// ---- 20_Product/10_BCF/11_Conv/15_Subsystem/10_Helper/F_GetSubSystemExternErrorData.TcPOU
FUNCTION F_GetSubSystemExternErrorData : ST_ErrorDataSet
(**************************************************************************************
 * 	Application		:	BoxControl Framework
 *	Revision		:	$Revision: 404529 $
 *	Revision date	:	$Date: 2018-04-23 08:21:38 +0200 (Mo., 23 Apr 2018) $
 *	Last changed by	:	$Author: b7bolm $
 *	URL				:	$URL: http://almscdc.swisslog.com/repo/SWPD/Development/BoxControlFramework/20_Release/trunk/01_Software/BCF/BCF/JumpStart/20_Product/10_App/15_Subsystem/10_Lib/10_Conv/10_Functions/F_GetSubSystemExternErrorData.TcPOU $
 *
 *	Purpose			:	Return subsystem error data
 *
 * ------------------------------------------------------------------------------------
 *	Copyright Swisslog [IP AG], Switzerland. All rights reserved.
 * 
 * ------------------------------------------------------------------------------------
 *	
 * 	Revision History: 
 *
 * 	VERSION			DATE			INITIALS			DESCRIPTION
 *	0.1				01.01.2001		swl					Example
 *
 **************************************************************************************)


// Check reference is valid
IF __ISVALIDREF(Subsystemregistry.rSubsystemData) THEN
	// Return error data
	F_GetSubSystemExternErrorData :=Subsystemregistry.rSubsystemData.ErrorData.ExternalError;
END_IF

END_FUNCTION

// ---- 20_Product/10_BCF/11_Conv/15_Subsystem/10_Helper/F_GetSubSystemInterface.TcPOU
FUNCTION F_GetSubsystemInterface : ST_SubsystemInterface
(**************************************************************************************
 * 	Application		:	BoxControl Framework
 *	Revision		:	$Revision: 404529 $
 *	Revision date	:	$Date: 2018-04-23 08:21:38 +0200 (Mo., 23 Apr 2018) $
 *	Last changed by	:	$Author: b7bolm $
 *	URL				:	$URL: http://almscdc.swisslog.com/repo/SWPD/Development/BoxControlFramework/20_Release/trunk/01_Software/BCF/BCF/JumpStart/20_Product/10_App/15_Subsystem/10_Lib/10_Conv/10_Functions/F_GetSubSystemInterface.TcPOU $
 *
 *	Purpose			:	Returns group interface
 *
 * ------------------------------------------------------------------------------------
 *	Copyright Swisslog [IP AG], Switzerland. All rights reserved.
 * 
 * ------------------------------------------------------------------------------------
 *	
 * 	Revision History: 
 *
 * 	VERSION			DATE			INITIALS			DESCRIPTION
 *	0.1				01.01.2001		swl					Example
 *
 **************************************************************************************)

// Get Master speed from subsystem
IF __ISVALIDREF(SubsystemRegistry.rSubsystem) THEN
	// Return Subsystem interface
	F_GetSubsystemInterface := SubsystemRegistry.rSubsystem.SubsystemInterface;
END_IF

END_FUNCTION

// ---- 20_Product/10_BCF/11_Conv/15_Subsystem/10_Helper/F_GetSubSystemSettings.TcPOU
FUNCTION F_GetSubsystemSettings : ST_CFG_Subsystem
(**************************************************************************************
 * 	Application		:	BoxControl Framework
 *	Revision		:	$Revision: 404529 $
 *	Revision date	:	$Date: 2018-04-23 08:21:38 +0200 (Mo., 23 Apr 2018) $
 *	Last changed by	:	$Author: b7bolm $
 *	URL				:	$URL: http://almscdc.swisslog.com/repo/SWPD/Development/BoxControlFramework/20_Release/trunk/01_Software/BCF/BCF/JumpStart/20_Product/10_App/15_Subsystem/10_Lib/10_Conv/10_Functions/F_GetSubSystemSettings.TcPOU $
 *
 *	Purpose			:	Returns group settings
 *
 * ------------------------------------------------------------------------------------
 *	Copyright Swisslog [IP AG], Switzerland. All rights reserved.
 * 
 * ------------------------------------------------------------------------------------
 *	
 * 	Revision History: 
 *
 * 	VERSION			DATE			INITIALS			DESCRIPTION
 *	0.1				01.01.2001		swl					Example
 *
 **************************************************************************************)
VAR
	SubsystemReg	: ST_SubsystemRegistryConv;
END_VAR


// Get Master speed from subsystem
IF __ISVALIDREF(SubsystemRegistry.rSettingsSubsystem) THEN
	// Return Subsystem settings
	F_GetSubsystemSettings := SubsystemRegistry.rSettingsSubsystem;
END_IF

END_FUNCTION

// ---- 20_Product/10_BCF/11_Conv/15_Subsystem/10_Helper/F_ResetExternalSubsystemError.TcPOU
FUNCTION F_ResetExternalSubsystemError : BOOL
(**************************************************************************************
 * 	Application		:	BoxControl Framework
 *	Revision		:	$Revision: 404529 $
 *	Revision date	:	$Date: 2018-04-23 08:21:38 +0200 (Mo., 23 Apr 2018) $
 *	Last changed by	:	$Author: b7bolm $
 *	URL				:	$URL: http://almscdc.swisslog.com/repo/SWPD/Development/BoxControlFramework/20_Release/trunk/01_Software/BCF/BCF/JumpStart/20_Product/10_App/15_Subsystem/10_Lib/10_Conv/10_Functions/F_ResetExternalSubsystemError.TcPOU $
 *
 *	Purpose			:	Reset external error
 *						Add an External error, which will be reported over the configured
 *						position.
 *						
 *
 * ------------------------------------------------------------------------------------
 *	Copyright Swisslog [IP AG], Switzerland. All rights reserved.
 * 
 * ------------------------------------------------------------------------------------
 *	
 * 	Revision History: 
 *
 * 	VERSION			DATE			INITIALS			DESCRIPTION
 *	0.1				01.01.2001		swl					Example
 *
 **************************************************************************************)
VAR_INPUT
	Reset			: BOOL;
END_VAR


IF __ISVALIDREF(SubsystemRegistry.rSubsystem) THEN
	// Reset external error on instance
	SubsystemRegistry.rSubsystem.M_ResetExternalError(
		mReset := Reset);
END_IF

END_FUNCTION

// ---- 20_Product/10_BCF/11_Conv/15_Subsystem/10_Helper/F_ResetSubsystemError.TcPOU
FUNCTION F_ResetSubsystemError : BOOL
(**************************************************************************************
 * 	Application		:	BoxControl Framework
 *	Revision		:	$Revision: 404529 $
 *	Revision date	:	$Date: 2018-04-23 08:21:38 +0200 (Mo., 23 Apr 2018) $
 *	Last changed by	:	$Author: b7bolm $
 *	URL				:	$URL: http://almscdc.swisslog.com/repo/SWPD/Development/BoxControlFramework/20_Release/trunk/01_Software/BCF/BCF/JumpStart/20_Product/10_App/15_Subsystem/10_Lib/10_Conv/10_Functions/F_ResetSubsystemError.TcPOU $
 *
 *	Purpose			:	Reset Subsystem error
 *
 * ------------------------------------------------------------------------------------
 *	Copyright Swisslog [IP AG], Switzerland. All rights reserved.
 * 
 * ------------------------------------------------------------------------------------
 *	
 * 	Revision History: 
 *
 * 	VERSION			DATE			INITIALS			DESCRIPTION
 *	0.1				01.01.2001		swl					Example
 *
 **************************************************************************************)

// Reset subsystem error
IF __ISVALIDREF(SubsystemRegistry.rSubsystem) THEN
	// Reset error on Subsystem
	SubsystemRegistry.rSubsystem.M_ResetError();
END_IF

END_FUNCTION

// ---- 20_Product/10_BCF/11_Conv/15_Subsystem/10_Helper/F_SetExternalSubsystemError.TcPOU
FUNCTION F_SetExternalSubsystemError : BOOL
(**************************************************************************************
 * 	Application		:	BoxControl Framework
 *	Revision		:	$Revision: 404529 $
 *	Revision date	:	$Date: 2018-04-23 08:21:38 +0200 (Mo., 23 Apr 2018) $
 *	Last changed by	:	$Author: b7bolm $
 *	URL				:	$URL: http://almscdc.swisslog.com/repo/SWPD/Development/BoxControlFramework/20_Release/trunk/01_Software/BCF/BCF/JumpStart/20_Product/10_App/15_Subsystem/10_Lib/10_Conv/10_Functions/F_SetExternalSubsystemError.TcPOU $
 *
 *	Purpose			:	Set external error
 *						Add an External error, which will be reported over the configured
 *						position.
 *						
 *
 * ------------------------------------------------------------------------------------
 *	Copyright Swisslog [IP AG], Switzerland. All rights reserved.
 * 
 * ------------------------------------------------------------------------------------
 *	
 * 	Revision History: 
 *
 * 	VERSION			DATE			INITIALS			DESCRIPTION
 *	0.1				01.01.2001		swl					Example
 *
 **************************************************************************************)
VAR_INPUT
	ErrorType		: E_ErrorType; // Error message type
	ErrorParam		: STRING(System.ERROR_PARAM_STRINGLENGTH); // Error parameter
	ErrorMsg		: INT; // Error message as String (Will be mapped to error code)
END_VAR


IF __ISVALIDREF(SubsystemRegistry.rSubsystem) THEN
	// Set external error on instance
	SubsystemRegistry.rSubsystem.M_SetExternalError(
		mErrorType 	:= ErrorType,
		mErrorParam := ErrorParam,
		mErrorCode 	:= ErrorMsg);
END_IF

END_FUNCTION

// ---- 20_Product/20_ProBox/10_Base/09_Overrides/FB_PB_FunctionConv.TcPOU
FUNCTION_BLOCK INTERNAL FB_PB_FunctionConv EXTENDS FB_FunctionConv
VAR_INPUT
END_VAR
VAR_OUTPUT
END_VAR

METHOD PROTECTED M_GetNextTransportData : REFERENCE TO ST_TransportData

VAR_INPUT
	mZoneNumber 	: INT; // Number of the zone
END_VAR

VAR
	NextFunction	: E_FunctionNumber;
	TempCopy		: E_FunctionNumber;
END_VAR

//Solves BCFD-11487 M_GetTransportData returns TransportData for wrong zone (in some situations)
//Solves BCFD-11583 HandoverState enters Active when next is Taking over from another function

//when Next function transport data is expected, we need to make sure that M_GetNextTransportData return correct data (Next -> Previus)
NextFunction := FunctionInterface.In.eNextFunctionNumber;
IF(__ISVALIDREF(FunctionRegistry[NextFunction].rFunctionInterface)) THEN
	TempCopy := FunctionRegistry[NextFunction].rFunctionInterface.In.eNextFunctionNumber;
	FunctionRegistry[NextFunction].rFunctionInterface.In.eNextFunctionNumber := E_FunctionNumber.F_BEGIN_FUNCTION;
	M_GetNextTransportData REF= SUPER^.M_GetNextTransportData(mZoneNumber);
	FunctionRegistry[NextFunction].rFunctionInterface.In.eNextFunctionNumber := TempCopy;
ELSE
	M_GetNextTransportData REF= SUPER^.M_GetNextTransportData(mZoneNumber);
END_IF
END_METHOD

METHOD PROTECTED M_GetPreviousTransportData: REFERENCE TO ST_TransportData

VAR_INPUT
	mZoneNumber 	: INT; // Number of the zone
END_VAR

VAR
	PrevFunction	: E_FunctionNumber;
	TempCopy		: E_FunctionNumber;
END_VAR

//Solves BCFD-11487 M_GetTransportData returns TransportData for wrong zone (in some situations)
//Solves BCFD-11583 HandoverState enters Active when next is Taking over from another function

//when previous function transport data is expected, we need to make sure that M_GetNextTransportData return correct data (prevous ->Next)
PrevFunction := FunctionInterface.In.ePrevFunctionNumber;
IF(__ISVALIDREF(FunctionRegistry[PrevFunction].rFunctionInterface)) THEN
	TempCopy := FunctionRegistry[PrevFunction].rFunctionInterface.In.ePrevFunctionNumber;
	FunctionRegistry[PrevFunction].rFunctionInterface.In.ePrevFunctionNumber := E_FunctionNumber.F_BEGIN_FUNCTION;
	M_GetPreviousTransportData REF= SUPER^.M_GetPreviousTransportData(mZoneNumber);
	FunctionRegistry[PrevFunction].rFunctionInterface.In.ePrevFunctionNumber := TempCopy;
ELSE
	M_GetPreviousTransportData REF= SUPER^.M_GetPreviousTransportData(mZoneNumber);
END_IF
END_METHOD

END_FUNCTION_BLOCK

// ---- 20_Product/20_ProBox/22_ProMove/03_Controls/02_TransportControl/FB_PB_TransportControlEmulation.TcPOU
FUNCTION_BLOCK FB_PB_TransportControlEmulation EXTENDS FB_TransportControlEmulation
(**************************************************************************************
 * 	Application		:	Pro Box
 *	Revision		:	$Revision:  $
 *	Revision date	:	$Date: $
 *	Last changed by	:	$Author: q8hedls $
 *	URL				:	$$
 *
 *	Purpose			:	Override BCF Transport control emulation
 *
 * ------------------------------------------------------------------------------------
 *	Copyright Swisslog [IP AG], Switzerland. All rights reserved.
 * 
 * ------------------------------------------------------------------------------------
 *	
 **************************************************************************************)
VAR_INPUT
	
END_VAR

VAR_IN_OUT
	//ZoneData				: ST_ZoneDataEmulation; // Zone data
END_VAR


SUPER^(ZoneData :=ZoneData);

END_FUNCTION_BLOCK

// ---- 20_Product/20_ProBox/22_ProMove/03_Controls/02_TransportControl/FB_ProBoxTransportControl.TcPOU
//ProBox transportcontroller
FUNCTION_BLOCK FB_ProBoxTransportControl EXTENDS FB_TransportControl
(**************************************************************************************
 * 	Application		:	ProBox
 *	Revision		:	$Revision:  $
 *	Revision date	:	$Date: $
 *	Last changed by	:	$Author: $
 *	URL				:	$URL: $
 *
 *	Purpose			:	The transport control is responsible for the coordinated
 *                      physical TU and logical data movement and ensures the relation
 *                      to the position for the ProMove Pallet system.
 *
 **************************************************************************************)
VAR_INPUT
	CtrlInPbTc				: ST_CtrlInPbTc;// Control input for Pro box Transport control
END_VAR
VAR	
	_PB_TransportCtrlData	: ST_PB_TransportCtrl;
	_ValidPrevFunction		: E_FunctionNumber;
	_ValidPrevZone			: INT;	
	_PbTcDebugLogLevel		: INT:=0; 		//ProBox Transport Control Debug level. 0 = Off, 1=States, 2 Verbose
END_VAR

VAR_TEMP
		
	PB_SimultaniousDisableTakeover		 :BOOL;	//TRUE = Release TU's
	PB_PreventTakeover					: BOOL; //For Multi Zone Functions
	PB_PreventHandover					: BOOL; //workaround for BCF transportcontroller not capable of handling a occupied after transition error
	PB_InhibitHandoverRun				: BOOL;	//Force stopping of drive
	PB_ForceTakeoverRun					: BOOL; //Force motor run of drive
	
	// internal variables only for debuging purposes
	PrevTrspState						: E_TransportState;
	PrevHandOvrState					: E_HandOverState;
	PrevTakeOvrState					: E_TakeOverState;		
END_VAR

IF(_PbTcDebugLogLevel>0) THEN
	// internal variables onlyfor debuging purposes
	PrevTrspState := ZoneData.TransportControlData.eTransportState;
	PrevHandOvrState := ZoneData.TransportControlData.eHandOverState;
	PrevTakeOvrState := ZoneData.TransportControlData.eTakeOverState;
END_IF

//---------------------------------------------------------------------------------------------------
// Init and checks for ProBox
//---------------------------------------------------------------------------------------------------
_M_PB_Init(ZoneData);
_M_InputMapping();


//---------------------------------------------------------------------------------------------------
// Pre-tasks that must be performed before runnign BCF transportcontrol
//---------------------------------------------------------------------------------------------------

_M_SyntheticSensor(ZoneData);
_M_GapCheck(ZoneData,ErrorData);
_M_PB_PreErrorCheck(ZoneData,ErrorData,PB_PreventTakeover,PB_PreventHandover);
_M_PB_PreTrspCtrl(ZoneData,ErrorData,PB_ForceTakeoverRun,PB_SimultaniousDisableTakeover,PB_PreventTakeover);

//---------------------------------------------------------------------------------------------------
// Call BCF TransportController
//---------------------------------------------------------------------------------------------------

TransportEnableTakeOver := TransportEnableTakeOver AND (NOT PB_SimultaniousDisableTakeover AND NOT PB_PreventTakeover);
TransportEnableHandOver := TransportEnableHandOver AND NOT PB_PreventHandover;
SUPER^(ZoneData:=ZoneData,ErrorData:=ErrorData);



//---------------------------------------------------------------------------------------------------
// Post-tasks that must be performed after BCF transportcontrol where executed
//---------------------------------------------------------------------------------------------------
_M_PB_PostTrspCtrl(ZoneData,PB_InhibitHandoverRun);
_M_PB_PostErrorCheck(ZoneData);
_M_PB_SpeedControl(ZoneData);

//PB transportcontrol controlling driving.
Outputs.DriveHandoverRun := (Outputs.DriveHandoverRun AND NOT PB_InhibitHandoverRun);
Outputs.DriveTakeoverRun := Outputs.DriveTakeoverRun OR PB_ForceTakeoverRun;

ZoneData.TransportControlData.Stopped := Param.rOperationState.eState = E_PositionState.STOPPED OR
									 	 Param.rOperationState.eState = E_PositionState.STOPPING AND NOT
									     DriveTakeoverRun AND NOT DriveHandoverRun;

//check RequestNext / DeleteNext and RequestPrev / DeletePrev
_M_ControlTransportRequests();



//---------------------------------------------------------------------------------------------------
// log transitions (To be deleted
//---------------------------------------------------------------------------------------------------
IF(_PbTcDebugLogLevel>0) THEN
	IF( PrevTrspState<>ZoneData.TransportControlData.eTransportState OR 
		PrevHandOvrState<>ZoneData.TransportControlData.eHandOverState OR
		PrevTakeOvrState<>ZoneData.TransportControlData.eTakeOverState) THEN
					DebugMsg := F_AddDividerToSisString(Param.rSettings.ZoneName);				
					DebugMsg := CONCAT(DebugMsg, '. Transport state: ');
					DebugMsg := CONCAT(DebugMsg, INT_TO_STRING(ZoneData.TransportControlData.eTransportState));
					DebugMsg := CONCAT(DebugMsg, '. Handover state: ');
					DebugMsg := CONCAT(DebugMsg, INT_TO_STRING(ZoneData.TransportControlData.eHandOverState));
					DebugMsg := CONCAT(DebugMsg, '. Takeover state: ');
					DebugMsg := CONCAT(DebugMsg, INT_TO_STRING(ZoneData.TransportControlData.eTakeOverState));
					DebugMsg := CONCAT(DebugMsg, '. HO Run: ');
					DebugMsg := CONCAT(DebugMsg, BOOL_TO_STRING(Outputs.DriveHandoverRun));
					DebugMsg := CONCAT(DebugMsg, '. TO Run: ');
					DebugMsg := CONCAT(DebugMsg, BOOL_TO_STRING(Outputs.DriveTakeoverRun));				
					fbDebugMsg.M_SendInfoMsg(DebugMsg);
	END_IF	
END_IF

//---------------------------------------------------------------------------------------------------
// Set error param with informative descriptions 
//---------------------------------------------------------------------------------------------------
//Only set the ErrorParam once, ie when the zone has no error. Also, do not override ErrorParam if there is text already set
IF(ZoneData.ErrorData.ErrorState <> E_ErrorState.ERROR AND ErrorData.ErrorParam[0]=0) THEN
	
	CASE ErrorData.ErrorCode.Conv OF 
		E_ErrorConv.TIMEOUT_TAKEOVER:
			ErrorData.ErrorParam	:= 'Takeover abnormal distance(TimeOut)';		
		E_ErrorConv.POSITION_OCCUPIED_BEFORE_TAKEOVER:
        	ErrorData.ErrorParam	:= 'Position occupied before takeover';
		E_ErrorConv.POSITION_OCCUPIED_AFTER_HANDOVER:
			ErrorData.ErrorParam	:= 'Position occupied after transmission';		
		E_ErrorConv.TU_DATA_SET_EMPTY_ZONE_OCCUPIED:
			ErrorData.ErrorParam	:= 'TU data set empty, position occupied'; 
  		E_ErrorConv.TU_DATA_SET_OCCUPIED_ZONE_FREE:
			ErrorData.ErrorParam	:= 'TU data set occupied, position free';	
		
	END_CASE
	
END_IF

METHOD PRIVATE _M_AllZonesOccupied : BOOL
VAR_INPUT
END_VAR

_M_AllZonesOccupied := _M_CountTus() = _PB_TransportCtrlData.NumberOfZones;
END_METHOD

METHOD PRIVATE _M_CheckZoneError : BOOL
VAR_INPUT
	eFunctionNumber		: E_FunctionNumber; // Function number
	ZoneNumber			: INT; // Zone number
END_VAR
// Check if function number and zone is valid
IF eFunctionNumber > E_FunctionNumber.F_BEGIN_FUNCTION AND
   eFunctionNumber < E_FunctionNumber.F_END_FUNCTION AND
   ZoneNumber > 0 AND ZoneNumber <= NUMBER_OF_ZONES_PER_FUNCTION THEN
  
   IF __ISVALIDREF(FunctionRegistry[eFunctionNumber].Zone[ZoneNumber].refZoneData) THEN
		// Zone errordata
		_M_CheckZoneError := FunctionRegistry[eFunctionNumber].Zone[ZoneNumber].refZoneData.ErrorData.Error.ErrorType = E_ErrorType.ERROR;
	END_IF
END_IF
END_METHOD

METHOD PRIVATE _M_ControlTransportRequests : BOOL
VAR_INPUT
END_VAR
//Disable fbRoutingServiceRetry waiting for RECALL_SERVICE_TIMEOUT ie 2S to request next function.
IF(SUPER^.Init AND  Param.rSettings.EnableRoutingUpdate AND _PB_TransportCtrlData.NumberOfZones>1 AND _PB_TransportCtrlData.IsFirstZone) THEN
	fbRoutingServiceRetry(IN := TRUE);
END_IF



//PB-6238 eNextFunctionNumber not set to F_BEGIN_FUNCTION after pallet removal
//request next function required when a zone is in state free.
IF(_PB_TransportCtrlData.NumberOfZones>1 AND _PB_TransportCtrlData.IsLastZone) THEN
	{warning disable C0371}
	IF( ZoneData.TransportControlData.eTransportState = E_TransportState.FREE) THEN		
		Outputs.DeleteNextTransportData:=TRUE;// request next
	END_IF
	{warning restore C0371}
END_IF


// control Delete next transportdata for multi zone functions. Don't delete next transport data unless finished handover
// fix for BCFD-11642 - TransportControl M_RequestPrev deletes previous on the same cycle as the transport starts
// -Also single zone functions needs to reset reqest signals
IF(Outputs.DeleteNextTransportData AND NOT Outputs.RequestNextTransportData) THEN
	//DeleteNextTransportData is requested	
	IF(_M_TransferBusy(Param.ZoneNumber,3)) THEN		
		Outputs.DeleteNextTransportData:=FALSE;	//Prevent delete next function			
	END_IF	
END_IF
IF(Outputs.DriveHandoverRun) THEN (*PB-5879 - TransportControl - TransportUnit transport error	AND BCFD-11642 - TransportControl M_RequestPrev deletes previous on the same cycle as the transport starts*)
	Outputs.DeleteNextTransportData:=FALSE;	//Prevent delete next function
	Outputs.RequestNextTransportData:=FALSE;//Prevent delete next function
END_IF

// control Delete prev transportdata for multi zone functions. Don't delete Prev transport data unless all zones finished takeover
// -Also single zone functions needs to reset reqest signals 
IF(Outputs.DeletePrevTransportData AND NOT Outputs.RequestPrevTransportData) THEN
	//DeletePrevTransportData is requested	
	IF(_M_TransferBusy(Param.ZoneNumber,1)) THEN
		Outputs.DeletePrevTransportData:=FALSE;	//Prevent delete previous function		
	END_IF			
END_IF
// fix for BCFD-11642 - TransportControl M_RequestPrev deletes previous on the same cycle as the transport starts
IF(Outputs.DriveTakeoverRun) THEN	
	Outputs.DeletePrevTransportData:=FALSE;	//Prevent delete previous function
	Outputs.RequestPrevTransportData:=FALSE;	//Prevent delete previous function
END_IF
END_METHOD

METHOD PRIVATE _M_CountTus : INT
VAR
	i,OccupiedCount:INT;
END_VAR
//Count TU's
FOR i:=1 TO _PB_TransportCtrlData.NumberOfZones DO
	IF(__ISVALIDREF(FunctionRegistry[Param.reFunctionNumber].Zone[i].refZoneData)) THEN
		IF(FunctionRegistry[Param.reFunctionNumber].Zone[i].refZoneData.TransportControlData.Occupied) THEN
			OccupiedCount := OccupiedCount + 1;
		END_IF
	END_IF
END_FOR
	
_M_CountTus:=OccupiedCount;
END_METHOD

METHOD PRIVATE _M_GapCheck : BOOL
VAR_IN_OUT
	ZoneData				: ST_ZoneData;
	ErrorData 				: ST_ErrorDataSet; // Error data 
END_VAR
VAR_INST		
	GapCheckState			: INT;			
	distanceMeter			: FB_DisplacementMeter();
	TestRunning	: BOOL;
END_VAR
VAR
	QuitTest				: BOOL;
END_VAR
IF(_PB_TransportCtrlData.NumberOfZones=1 OR NOT _PB_TransportCtrlData.IsLastZone) THEN
	RETURN;
END_IF


//Escape test
QuitTest := ZoneData.TransportControlData.eTransportState <> E_TransportState.SIMULTANEOUS AND
			ZoneData.TransportControlData.eTransportState <> E_TransportState.SIMULTANEOUS_STOP; 

CASE  GapCheckState OF
	0:		
		//Start test
		IF( ZoneData.TransportControlData.eTakeOverState = E_TakeOverState.ACTIVE AND
			ZoneData.TransportControlData.eTransportState = E_TransportState.SIMULTANEOUS) THEN			
			GapCheckState := GapCheckState+1;
			TestRunning:=FALSE;
		END_IF
	1:
		//check time when sensor detects gap of rear edge
		IF(NOT ZoneOccupied) THEN
			TestRunning:=TRUE;
			GapCheckState := GapCheckState+1;			
		ELSIF(QuitTest) THEN
			GapCheckState:=0;
		END_IF
		
	2: //Check when new pallet arrives
		IF(ZoneOccupied) THEN
			IF(distanceMeter.Q) THEN				 
				GapCheckState := GapCheckState+1; //Test successful				
			ELSE
				GapCheckState :=4; //error state				
			END_IF
		ELSIF(QuitTest) THEN
			GapCheckState := GapCheckState+1;
		END_IF 
	
	3:	
		//wait for Escape test to occure.
		IF(QuitTest) THEN			
			GapCheckState:=0;
		END_IF 
	4:
		//error
		F_SetError(	
					ErrorType	:= E_ErrorType.ERROR,
					ErrorParam	:= 'Gap not detected',
					ErrorMsg	:= E_ErrorConv.GAP_CHECK_ACTIVE,
					ErrorData	:= ErrorData);		
					
		//recover from error. sensor needs to be un-occupied. (or should it be enought with just a acknowledge of error?)
		IF(NOT ZoneOccupied) THEN
			GapCheckState:=0;
		END_IF
		
END_CASE


distanceMeter(
	Run:=TestRunning, 
	EncoderValueInc:=SUPER^.EncoderValue,
	MaxEncoderValueInc 	:= SUPER^.MaxEncoderValue, 
	RateIncPerMM:=1,
	SetPoint := 100 (*mm*));
END_METHOD

METHOD PRIVATE _M_InputMapping : BOOL
VAR_INPUT
END_VAR
VAR
	ElementNumber : E_ElementNumber;
END_VAR

//Prerequsities for ProBox transports
IF(Param.rSettings.EnableMFC) THEN
	//Following parameters must have defined state in order for ProBox to guarantee known functionality
	Param.rSettings.EnableFreeRun := FALSE;
	Param.rSettings.EnableMultizone := FALSE;
	Param.rSettings.EnableJamAutoReset := FALSE;
	Param.rSettings.ClearingDistance := 0;
	Param.rSettings.AddTU_Data := FALSE;
	Param.rSettings.DeleteTU_DataTakeOver := FALSE;
	Param.rSettings.DeleteTU_DataZoneFree := FALSE;
	Param.rSettings.EnablePrestart:=FALSE;				//important to set to false for transfer units
	Param.rSettings.EnableRoutingUpdate:=TRUE;			//Default ON
END_IF

//Transport control Inputs
EnableFastSpeed:=FALSE;			//Probox needs an alternative way of treating low speeds than BCF transport control. (this functionality is always enabled, but the EnableFastSpeed is set to false so that the BCF transport controller shall not run code unnecessary


IF(__ISVALIDREF(FunctionRegistry[Param.reFunctionNumber].rFunctionInterface)) THEN
	IF(NOT FunctionRegistry[Param.reFunctionNumber].rFunctionInterface.In.FunctionEnable) THEN
		TransportEnableHandOver := FALSE;
		IF(_M_CountTus()=0 AND _PB_TransportCtrlData.IsFirstZone) THEN 
			TransportEnableTakeOver:=FALSE; //Disable takeover if all zones are free
		END_IF 
		TransportEnableHandOver:=FALSE; //disable handover for all zones
	END_IF
END_IF


IF(__ISVALIDREF(FunctionRegistry[Param.reFunctionNumber].rSettingsFunction)) THEN
	ElementNumber := FunctionRegistry[Param.reFunctionNumber].rSettingsFunction.eElementLink;
	IF(__ISVALIDREF(ElementRegistry[ElementNumber].rElementInterface)) THEN
		IF(NOT ElementRegistry[ElementNumber].rElementInterface.In.ElementEnable) THEN			
			IF(_M_CountTus()=0 AND _PB_TransportCtrlData.IsFirstZone) THEN 
				TransportEnableTakeOver:=FALSE; //Disable takeover if all zones are free
			END_IF
			TransportEnableHandOver:=FALSE; //disable handover for all zones
		END_IF	
	END_IF
END_IF
END_METHOD

// Check if zone is deslugging 
METHOD PRIVATE _M_IsDeslugging : BOOL
VAR_INPUT
END_VAR
VAR
	NextNumberOfZones : INT;
	MeNumberOfZones : INT;
	OccupiedCount:INT;
	IsLastZone : BOOL;
END_VAR

//Last zone shall check if deslugging
IF(NOT _PB_TransportCtrlData.IsLastZone) THEN
	RETURN;
END_IF

// Check if function number is valid
IF NextTransportData.eFunctionNumber > E_FunctionNumber.F_BEGIN_FUNCTION AND
   NextTransportData.eFunctionNumber < E_FunctionNumber.F_END_FUNCTION THEN
  	
	IF __ISVALIDREF(FunctionRegistry[NextTransportData.eFunctionNumber].rSettingsFunction) THEN   		
   		NextNumberOfZones := FunctionRegistry[NextTransportData.eFunctionNumber].rSettingsFunction.NumberOfZones;
	ELSE
		RETURN;		 
	END_IF
	
			
	//Count TU's on own function
	OccupiedCount := _M_CountTus();
			
	// Deslugging whait with handover last TU until next function has filled upp all zones.  
	_M_IsDeslugging := NextNumberOfZones < _PB_TransportCtrlData.NumberOfZones AND (OccupiedCount + NextNumberOfZones <= _PB_TransportCtrlData.NumberOfZones); 
	
END_IF
END_METHOD

METHOD _M_PB_Init : BOOL
VAR_IN_OUT
	ZoneData					: ST_ZoneData;
END_VAR

IF( NOT ZoneData.Init) THEN
	_PB_TransportCtrlData.Init:=FALSE;		
END_IF

IF(NOT _PB_TransportCtrlData.Init) THEN
	IF __ISVALIDREF(FunctionRegistry[Param.reFunctionNumber].rSettingsFunction) THEN   		
   		_PB_TransportCtrlData.NumberOfZones := FunctionRegistry[Param.reFunctionNumber].rSettingsFunction.NumberOfZones;
		_PB_TransportCtrlData.Init := TRUE; 
	END_IF
	//Set to Default value.
	MaxEncoderValue	:= 16#FFFF;
	
ELSE
	//For each call check following.
	IF __ISVALIDREF(FunctionRegistry[Param.reFunctionNumber].rSettingsFunction) THEN

		_PB_TransportCtrlData.IsFirstZone := (Param.ZoneNumber = 1 AND  FunctionRegistry[Param.reFunctionNumber].rSettingsFunction.FlowDirectionREV = FALSE) OR
											 (Param.ZoneNumber = _PB_TransportCtrlData.NumberOfZones AND  FunctionRegistry[Param.reFunctionNumber].rSettingsFunction.FlowDirectionREV = TRUE);   		
   		
		_PB_TransportCtrlData.IsLastZone := (Param.ZoneNumber = 1 AND  FunctionRegistry[Param.reFunctionNumber].rSettingsFunction.FlowDirectionREV = TRUE) OR
											 (Param.ZoneNumber = _PB_TransportCtrlData.NumberOfZones AND  FunctionRegistry[Param.reFunctionNumber].rSettingsFunction.FlowDirectionREV = FALSE);
		
		_PB_TransportCtrlData.LastZoneIx := SEL(NOT FunctionRegistry[Param.reFunctionNumber].rSettingsFunction.FlowDirectionREV ,1,_PB_TransportCtrlData.NumberOfZones);
   		_PB_TransportCtrlData.FirstZoneIx:= SEL(NOT FunctionRegistry[Param.reFunctionNumber].rSettingsFunction.FlowDirectionREV ,_PB_TransportCtrlData.NumberOfZones,1);
	ELSE
		; //raise error?
	END_IF	
END_IF
END_METHOD

METHOD PRIVATE _M_PB_PostErrorCheck : BOOL
VAR_IN_OUT
	ZoneData				: ST_ZoneData;
END_VAR


//error handling
CASE ZoneData.TransportControlData.eTransportState OF


	E_TransportState.OCCUPIED, E_TransportState.SIMULTANEOUS_OCCUPIED:
		IF( (Zonedata.TransportControlData.eTakeOverState = E_TakeOverState.COMPLETE OR Zonedata.TransportControlData.eTakeOverState = E_TakeOverState.INTERRUPTED) AND						 
			PrevTransportData.rTransportControlData.eHandOverState = E_HandOverState.STOP) THEN
			
			//Set takeover to interupted.
			Zonedata.TransportControlData.eTakeOverState := E_TakeOverState.INTERRUPTED;
		END_IF
			
END_CASE
END_METHOD

METHOD _M_PB_PostTrspCtrl : BOOL
VAR_INPUT
END_VAR
VAR_IN_OUT
	ZoneData			: ST_ZoneData;
	InhibitHandoverRun	: BOOL;	
END_VAR

InhibitHandoverRun:=FALSE;


CASE ZoneData.TransportControlData.eTransportState OF
	E_TransportState.TAKEOVER:		
		//adjust takeover distance on last zone, since the takeover may start earlier than the zone is. (depending on zone length configuration)
		//when running without MFC the plausability check must be intact, hence, adjusting the zone length		
		IF(_PB_TransportCtrlData.NumberOfZones>1 AND _PB_TransportCtrlData.IsLastZone AND			
			ZoneData.TransportControlData.eTakeOverState = E_TakeOverState.ACTIVE AND
			F_PB_GetTransportControlDataRef(Param.reFunctionNumber,_PB_TransportCtrlData.FirstZoneIx).eTransportState = E_TransportState.SIMULTANEOUS) THEN
			// Reset timeout take
			fbTimeoutTake(RUN:=FALSE); //reset DisplacmentDistance in order to adjust the correct takeover length
		END_IF
 

	E_TransportState.OCCUPIED, E_TransportState.HANDOVER:
		
		//if previous is occupied and we should start slugging, this happens when adding pallets by TTA or chaning drive direction
		//should be fixed in BCF transportControl in state occupied.
		IF( ((_PB_TransportCtrlData.IsFirstZone AND CtrlInPbTc.EnableSlugging) OR 
			 (NOT _PB_TransportCtrlData.IsFirstZone AND PrevTransportData.rTransportControlData.Occupied)) AND
			Param.rSettings.EnableSimultaneousTransport AND ZoneData.TransportControlData.Occupied AND 
			ZoneData.TransportControlData.NumberOfPresentTUs>0 AND TU_DataTable[ZoneData.TransportControlData.TU_DataIndex].DataSet.JobPresent) THEN			
			 ZoneData.TransportControlData.eTransportState := E_TransportState.SIMULTANEOUS_OCCUPIED;
			 ZoneData.TransportControlData.eHandOverState := E_HandOverState.IDLE;
			 IF(_PbTcDebugLogLevel>1) THEN fbDebugMsg.M_SendInfoMsg('Force state to SIMULTANEOUS_OCCUPIED'); END_IF			 
		END_IF
					
	E_TransportState.SIMULTANEOUS_OCCUPIED:
		//Deslugging must stop conveyor at last zone if next zone is longer than own zone	 
		IF(Outputs.DriveHandoverRun AND ZoneData.TransportControlData.eHandOverState = E_HandOverState.COMPLETE AND _M_IsDeslugging()) THEN 
			InhibitHandoverRun:=TRUE;//Outputs.DriveHandoverRun :=FALSE;
		END_IF
END_CASE
END_METHOD

METHOD PRIVATE _M_PB_PreErrorCheck : BOOL
VAR_IN_OUT
	ZoneData					: ST_ZoneData;
	ErrorData 					: ST_ErrorDataSet; // Error data	
	PreventTakeover				: BOOL;
	PreventHandover				: BOOL;
END_VAR
VAR_INST
	Error_181					: BOOL; //Error Position occupied after handover
END_VAR

(*IF(NOT _PB_TransportCtrlData.Init AND NOT Param.rSettings.EnableMFC) THEN
	F_SetError(	
			ErrorType	:= E_ErrorType.WARNING,
			ErrorParam	:= 'MFC has to be enabled for ProBox transport control',
			ErrorMsg	:= E_ErrorConv.CONFIGURATION_ERROR,
			ErrorData	:= ErrorData);
END_IF*)


//error handling
CASE ZoneData.TransportControlData.eTransportState OF

	E_TransportState.OCCUPIED, E_TransportState.SIMULTANEOUS_OCCUPIED:
		//Keep TU Data on last zone if first zone not finalized takeover
		IF( _PB_TransportCtrlData.IsLastZone AND 
			NOT F_PB_GetTransportControlDataRef(Param.reFunctionNumber, _PB_TransportCtrlData.FirstZoneIx).Occupied AND
			F_PB_GetTransportControlDataRef(Param.reFunctionNumber, _PB_TransportCtrlData.FirstZoneIx).NumberOfPresentTUs>0) THEN
 				PreventHandover:=TRUE;
		END_IF
		
		//error handling when previous has error.
		IF( (Zonedata.TransportControlData.eTakeOverState = E_TakeOverState.COMPLETE OR Zonedata.TransportControlData.eTakeOverState = E_TakeOverState.INTERRUPTED) AND
			//_M_CheckZoneError(_ValidPrevFunction,_ValidPrevZone)) THEN						 
			PrevTransportData.rTransportControlData.eHandOverState = E_HandOverState.STOP) THEN
			//If prev has error 181 (POSITION_OCCUPIED_AFTER_HANDOVER) then set takeover interupted.			
			IF(_PbTcDebugLogLevel>1 AND Zonedata.TransportControlData.eTakeOverState <> E_TakeOverState.INTERRUPTED) THEN 
				fbDebugMsg.M_SendInfoMsg('Prev has error POSITION_OCCUPIED_AFTER_HANDOVER');
			END_IF
			Zonedata.TransportControlData.eTakeOverState := E_TakeOverState.INTERRUPTED;
			PreventHandover:=TRUE;		
			
			// Set error to stop transfer when slugging (create train) when previous has error 'POSITION_OCCUPIED_AFTER_HANDOVER'
			IF(_PB_TransportCtrlData.IsFirstZone AND _PB_TransportCtrlData.NumberOfZones>1 AND CtrlInPbTc.SlugSensorExists AND
				ZoneData.TransportControlData.eTransportState = E_TransportState.SIMULTANEOUS_OCCUPIED) THEN				
				F_SetError(	
					ErrorType	:= E_ErrorType.ERROR,
					ErrorParam	:= 'Check Slug Sensor',
					ErrorMsg	:= E_ErrorConv.TRANSFER_ERROR,
					ErrorData	:= ErrorData);
			END_IF
		
		//recover			
		ELSIF( Zonedata.TransportControlData.eTakeOverState = E_TakeOverState.INTERRUPTED AND
			PrevTransportData.rTransportControlData.eHandOverState <> E_HandOverState.STOP) THEN
			Zonedata.TransportControlData.eTakeOverState := E_TakeOverState.COMPLETE;
		END_IF
		Error_181:=FALSE;
				 
		
		
	E_TransportState.TAKEOVER:
			
		//Error check that is missing in BCF TransportControl when EnableSimultaneousTranspor is enabled 
		IF( PrevTransportData.rTransportControlData.eHandOverState = E_HandOverState.READY AND ZoneOccupied AND Param.rSettings.EnableSimultaneousTransport) THEN				
			// Set error
			F_SetError(	
				ErrorType	:= E_ErrorType.ERROR,
				ErrorParam	:= '',
				ErrorMsg	:= E_ErrorConv.POSITION_OCCUPIED_BEFORE_TAKEOVER,
				ErrorData	:= ErrorData);
		END_IF
		
		//First zone shall check last sensor (for multi zone functions) regardless if EnableSimultaneousTransport is enabled or not before taking over, and all zones are free (un-occupied). 
		IF(_PB_TransportCtrlData.IsFirstZone AND _PB_TransportCtrlData.NumberOfZones>1 AND 
			PrevTransportData.rTransportControlData.eHandOverState = E_HandOverState.READY) THEN
			
			IF(_M_CountTus() = 0 AND CtrlInPbTc.StopSensor) THEN //F_PB_GetTransportControlDataRef(Param.reFunctionNumber, _PB_TransportCtrlData.LastZoneIx).SensorOccupied) THEN				
				// Set error (should be on last zone or on function level)				 
				F_SetError(	
					ErrorType	:= E_ErrorType.ERROR,
					ErrorParam	:= 'Last zone is occupied before takeover',
					ErrorMsg	:= E_ErrorConv.POSITION_OCCUPIED_BEFORE_TAKEOVER,
					ErrorData	:= ErrorData);
				//ihibit takeover
				PreventTakeover := TRUE;				
			END_IF
		END_IF
	
	
	E_TransportState.HANDOVER:
		//Correction of BCF Transport control, since Position occupied after handover error (181) is possible to acknowledge and proceed.
		IF(ErrorData.ErrorCode.Conv=E_ErrorConv.POSITION_OCCUPIED_AFTER_HANDOVER)THEN
			Error_181:=TRUE;
		END_IF
		IF(ZoneOccupied AND Error_181) THEN
			F_SetError(	
					ErrorType	:= E_ErrorType.ERROR,
					ErrorParam	:= '',
					ErrorMsg	:= E_ErrorConv.POSITION_OCCUPIED_AFTER_HANDOVER,
					ErrorData	:= ErrorData);
		ELSIF(NOT ZoneOccupied AND Error_181) THEN
			Error_181:=FALSE;
		END_IF
	
END_CASE
END_METHOD

METHOD PRIVATE _M_PB_PreTrspCtrl : BOOL
VAR_INPUT
END_VAR
VAR_IN_OUT
	ZoneData					: ST_ZoneData;
	ErrorData 					: ST_ErrorDataSet; // Error data
	ForceTakeoverRun			: BOOL;
	SimultaniousDisableTakeover : BOOL;
	PreventTakeover				: BOOL;	
END_VAR
DriveFeedInRun:=FALSE;	//Set default to False, due to bug in BCF transportcontrol (when group is in manual mode DriveFeedInRun is not canceled)

//Get previous function and zone
IF(ZoneData.TransportControlData.eTakeOverState = E_TakeOverState.ACTIVE) THEN
	IF(__ISVALIDREF(PrevTransportData.rTransportControlData)) THEN
		IF(PrevTransportData.eFunctionNumber <> E_FunctionNumber.F_BEGIN_FUNCTION) THEN
			_ValidPrevFunction 	:= PrevTransportData.eFunctionNumber;
			_ValidPrevZone		:= PrevTransportData.ZoneNumber;
		END_IF
	END_IF
		
END_IF

//ProBox Transport control multizone functionality
CASE ZoneData.TransportControlData.eTransportState OF

		
	E_TransportState.FREE, E_TransportState.TAKEOVER:
		
		//prevent multizone function to takeover on first zone(if empty) if any other zones are occupied
		IF(ZoneData.TransportControlData.eTakeOverState = E_TakeOverState.READY OR Zonedata.TransportControlData.eTakeOverState = E_TakeOverState.IDLE) THEN
			IF(_PB_TransportCtrlData.IsFirstZone AND _M_CountTus()>0) THEN
				PreventTakeover := TRUE;
			END_IF
			
		//recover from error previous occupied after transition  
		ELSIF(ZoneData.TransportControlData.Occupied AND
			  ZoneData.TransportControlData.eTakeOverState = E_TakeOverState.INTERRUPTED AND 
			  PrevTransportData.rTransportControlData.eHandOverState = E_HandOverState.ACTIVE) THEN
			  Zonedata.TransportControlData.eTakeOverState := E_TakeOverState.COMPLETE;			
		END_IF	
				

	E_TransportState.OCCUPIED:
		//solves issue when removing an TU from the system (InOutFeedAddon or CraneXover etc)
		IF(NOT ZoneData.TransportControlData.Occupied AND ZoneData.TransportControlData.NumberOfPresentTUs=0 AND NOT DriveRunning) THEN
			ZoneData.TransportControlData.eTransportState := E_TransportState.FREE; 
			IF(_PbTcDebugLogLevel>1) THEN fbDebugMsg.M_SendInfoMsg('Not logically occupied anymore'); END_IF
		END_IF

	
	E_TransportState.SIMULTANEOUS_OCCUPIED:
						
		//check if previous function is able to handover a TU when an simultanious takeover is complete in order to make possible to handover TU
		IF((ZoneData.TransportControlData.eTakeOverState = E_TakeOverState.READY OR Zonedata.TransportControlData.eTakeOverState = E_TakeOverState.IDLE) AND
			ZoneData.TransportControlData.eHandOverState <> E_HandOverState.COMPLETE AND F_PB_GetTransportControlDataRef(_ValidPrevFunction,_ValidPrevZone).eTransportState <> E_TransportState.SIMULTANEOUS_STOP) THEN
			
			//solves issue when removing an TU from the system (InOutFeedAddon or CraneXover etc)			
			IF(NOT ZoneData.TransportControlData.Occupied AND ZoneData.TransportControlData.NumberOfPresentTUs=0 AND NOT DriveRunning) THEN
				ZoneData.TransportControlData.eTransportState := E_TransportState.FREE;
				IF(_PbTcDebugLogLevel>1) THEN fbDebugMsg.M_SendInfoMsg('Not logically occupied anymore'); END_IF 
			
			
			//Control slugging
			ELSIF(_PB_TransportCtrlData.IsFirstZone AND CtrlInPbTc.EnableSlugging) THEN
				//Hold TU on first zone while creating train
				; // do nothing. SimultaniousDisableTakeover:=FALSE;
			ELSIF(_PB_TransportCtrlData.IsFirstZone AND _PB_TransportCtrlData.NumberOfZones>1 AND _M_AllZonesOccupied() AND NOT CtrlInPbTc.EnableSlugging) THEN
				SimultaniousDisableTakeover:=TRUE;
				IF(_PbTcDebugLogLevel>2) THEN fbDebugMsg.M_SendInfoMsg('Simultanious all zone occupied relese train'); END_IF
							
			ELSIF(_PB_TransportCtrlData.IsFirstZone AND _PB_TransportCtrlData.NumberOfZones>1 AND _ValidPrevFunction <> E_FunctionNumber.F_BEGIN_FUNCTION AND 
				 (F_PB_GetTransportControlDataRef(_ValidPrevFunction,_ValidPrevZone).eTransportState = E_TransportState.SIMULTANEOUS OR 
				  F_PB_GetTransportControlDataRef(_ValidPrevFunction,_ValidPrevZone).eHandOverState = E_HandOverState.COMPLETE)) THEN				
				ForceTakeoverRun:=TRUE;	//run conveoyr while previous is takeover acitve (else the TU's will stop when zone is occupied for a short while)
				
				IF(CtrlInPbTc.StopSensor) THEN
					F_SetError(	
						ErrorType	:= E_ErrorType.ERROR,
						ErrorParam	:= 'Slugging error, stop sensor covered',
						ErrorMsg	:= E_ErrorConv.TRANSFER_ERROR,
						ErrorData	:= ErrorData);	 		
				END_IF
				
			ELSIF(PrevTransportData.eFunctionNumber<>E_FunctionNumber.F_BEGIN_FUNCTION AND NOT PrevTransportData.rTransportControlData.Occupied AND
				 (PrevTransportData.rTransportControlData.NumberOfPresentTUs=0 OR _PB_TransportCtrlData.IsFirstZone)) THEN				   
				SimultaniousDisableTakeover:=TRUE;
				IF(_PbTcDebugLogLevel>2) THEN fbDebugMsg.M_SendInfoMsg('Simultanious relese train'); END_IF
			ELSIF(PrevTransportData.eFunctionNumber=E_FunctionNumber.F_BEGIN_FUNCTION) THEN
				SimultaniousDisableTakeover :=TRUE;	
				IF(_PbTcDebugLogLevel>2) THEN fbDebugMsg.M_SendInfoMsg('Previous not defined'); END_IF
			END_IF
		END_IF
				

	E_TransportState.HANDOVER:
		IF(ZoneData.TransportControlData.Occupied = FALSE AND ZoneData.TransportControlData.eHandOverState <> E_HandOverState.STOP) THEN
			//Solves PB-3889 - Stuck In Handover mode								
			ZoneData.TransportControlData.eTransportState := E_TransportState.FREE;			
		END_IF	
		
		//If handover and next function is complete, then always delete Occupied and NumberOfPresentTUs
		//-If the transfer has finished, but not if it where just started.
		//Solves issue with error 181=(POSITION_OCCUPIED_AFTER_HANDOVER) when Sensor is occupied after an complete handover, (A new handover is started after the error is acknowledged, despite theres no TU ID index or sensor occupied etc.)
		//Solves issue with creating ghost pallets.
		IF( NextTransportData.rTransportControlData.eTakeOverState = E_TakeOverState.COMPLETE AND ZoneData.TransportControlData.TU_DataIndex=0 AND
			ZoneData.TransportControlData.eHandOverState <> E_HandOverState.STOP) THEN
			ZoneData.TransportControlData.Occupied := FALSE;
			ZoneData.TransportControlData.NumberOfPresentTUs := 0;
		END_IF	
	
	E_TransportState.SIMULTANEOUS_STOP:		
				
			// If function is started
			IF Param.rOperationState.eState = E_PositionState.STARTED THEN
				// If transport is enabled
				IF Inputs.Enable.Transport THEN		
					// If no error is active
					IF ErrorData.ErrorType <> E_ErrorType.ERROR THEN
						
						IF(ZoneData.TransportControlData.NumberOfPresentTUs = 0 AND NOT ZoneData.TransportControlData.Occupied) THEN
							ZoneData.TransportControlData.eTransportState := E_TransportState.FREE;
						ELSE
							// Resume to simultaneous transport, otherwise do handover
							ZoneData.TransportControlData.eTransportState := E_TransportState.SIMULTANEOUS;
						END_IF						
					END_IF
				END_IF
			END_IF		
		
	
END_CASE
END_METHOD

METHOD PRIVATE _M_PB_SpeedControl : BOOL
VAR_INPUT
END_VAR
VAR_IN_OUT
	ZoneData					: ST_ZoneData;
END_VAR
//---------------------------------------------------------------------------------------------------
// ProBox Speed control
//---------------------------------------------------------------------------------------------------
// Reset fast speed active
ZoneData.TransportControlData.FastSpeedActive := FALSE;
// Set fast speed active
IF CurrentSpeed <> E_ProBoxMotorSpeed.CREEP_SPEED AND CurrentSpeed <> E_ProBoxMotorSpeed.LOW_SPEED THEN
	ZoneData.TransportControlData.FastSpeedActive := TRUE;
END_IF
// Reset fast speed active
IF NOT NextTransportData.rTransportControlData.FastSpeedActive AND Outputs.DriveHandoverRun THEN
	ZoneData.TransportControlData.FastSpeedActive := FALSE;
END_IF
END_METHOD

//Creats ZoneOccupied signal that is used by BCF transport control for Zones that does not have HW sensors.
METHOD PRIVATE _M_SyntheticSensor : BOOL
VAR_IN_OUT
	ZoneData					: ST_ZoneData;
END_VAR

VAR_INST	
	PrevZoneOccupiedRTrig			: R_TRIG;
	LastZoneOccupiedRTrig			: R_TRIG;
	
END_VAR

VAR
	//FirstZoneIx : INT:=1;
END_VAR
//Use stop sensor from CtrlInPbTc
IF(_PB_TransportCtrlData.NumberOfZones<=1) THEN	
	//set zone occupied when any sensor is active for elements with only one zone
		ZoneOccupied := CtrlInPbTc.SlugSensor OR CtrlInPbTc.StopSensor;
	RETURN;
ELSIF(_PB_TransportCtrlData.IsFirstZone AND CtrlInPbTc.SlugSensorExists) THEN
	
	//disable plausibile takeover filtering if Param.rSettings.TakeoverPlausibilityDistance = 0 (else BCF transport control will use pre defined value)
	IF(ZoneData.TransportControlData.eTakeOverState = E_TakeOverState.ACTIVE AND Param.rSettings.TakeoverPlausibilityDistance>0 AND NOT fbTakeoverPlausible.Q) THEN
		ZoneOccupied:=ZoneData.TransportControlData.Occupied;
		RETURN;	
	ELSE
		ZoneOccupied := CtrlInPbTc.SlugSensor;	
		RETURN;
	END_IF
	
ELSIF(_PB_TransportCtrlData.IsLastZone) THEN
	ZoneOccupied := CtrlInPbTc.StopSensor;
	RETURN;
END_IF

//only zones that does not have HW sensor shall execute following code

//Clear Zone occupied
IF(ZoneData.TransportControlData.eHandOverState = E_HandOverState.ACTIVE) THEN
	ZoneOccupied := FALSE;
END_IF


//Set ZoneOccupied depending on previous and next being occupied or not
//Note, the first zone taking over last TU from previous, must run entire TransportParam.ZoneLength so we know it is fully on the takeover conveyor.  
PrevZoneOccupiedRTrig(CLK:=PrevTransportData.rTransportControlData.Occupied AND PrevTransportData.rTransportControlData.eTransportState <> E_TransportState.HANDOVER AND PrevTransportData.eFunctionNumber<>E_FunctionNumber.F_BEGIN_FUNCTION);	
LastZoneOccupiedRTrig(CLK:=CtrlInPbTc.StopSensor AND (ZoneData.TransportControlData.eTransportState = E_TransportState.SIMULTANEOUS OR
													  ZoneData.TransportControlData.eTransportState = E_TransportState.SIMULTANEOUS_OCCUPIED));

IF(fbTimeoutTake.Run) THEN
	//ZoneLenght distance is achieved
	IF(fbTimeoutTake.Displacement > (TransportParam.ZoneLength-TransportParam.ZoneEndLength)) THEN
		IF(_PbTcDebugLogLevel>1 AND NOT ZoneOccupied) THEN fbDebugMsg.M_SendInfoMsg(CONCAT('Takeover Distance achieved: ', DINT_TO_STRING(fbTimeoutTake.Displacement))); END_IF  
		ZoneOccupied := TRUE;
	ELSIF(PrevZoneOccupiedRTrig.Q AND fbTimeoutTake.Displacement>0) THEN
		IF(_PbTcDebugLogLevel>1 AND NOT ZoneOccupied) THEN fbDebugMsg.M_SendInfoMsg(CONCAT('Takeover aborted PrevRTrig, distance: ', DINT_TO_STRING(fbTimeoutTake.Displacement))); END_IF
		ZoneOccupied := TRUE;	
	ELSIF(LastZoneOccupiedRTrig.Q) THEN
		IF(_PbTcDebugLogLevel>1 AND NOT ZoneOccupied) THEN fbDebugMsg.M_SendInfoMsg(CONCAT('Takeover aborted NextRTrig, distance: ', DINT_TO_STRING(fbTimeoutTake.Displacement))); END_IF
		ZoneOccupied := TRUE;
	END_IF
END_IF



// support TTA, TTC for zones that does not have HW sensors
IF(NOT ZoneData.Init) THEN	
	IF(ZoneData.TransportControlData.DataPresent AND ZoneData.TransportControlData.TU_DataIndex>0(*AND HW_SensorStop*)) THEN
		//Enable Adding TU when receiving TTA (*only possible if last zone is occupied*)
		ZoneOccupied:=TRUE;
	ELSIF(NOT ZoneData.TransportControlData.DataPresent AND ZoneData.TransportControlData.TU_DataIndex=0) THEN 
		//Clear SoftSensorOccupied on init of zone	// Clear SoftSensorOccupied uppon an init (TDQ)
		ZoneOccupied:=FALSE;
	END_IF
END_IF
END_METHOD

METHOD PRIVATE _M_TransferBusy : BOOL
VAR_INPUT
	MyZoneIx		: INT;
	TransferType	: UINT; //TakeOver=1, //HandOver=2, // Both=3	
END_VAR
VAR
	i	:INT;
	ToBusy,HoBusy	:BOOL;			
END_VAR

IF(_PB_TransportCtrlData.NumberOfZones<=1) THEN
	RETURN;
END_IF

//Check other zones transfer is busy or stopped/interupted
FOR i:=1 TO _PB_TransportCtrlData.NumberOfZones DO	
	IF(__ISVALIDREF(FunctionRegistry[Param.reFunctionNumber].Zone[i].refZoneData)) THEN
		IF(i<>MyZoneIx) THEN		
			IF(TransferType.0) THEN	// TransferType =1 or 3		 
				ToBusy := FunctionRegistry[Param.reFunctionNumber].Zone[i].refZoneData.TransportControlData.eTakeOverState <> E_TakeOverState.IDLE AND 
						  FunctionRegistry[Param.reFunctionNumber].Zone[i].refZoneData.TransportControlData.eTakeOverState <> E_TakeOverState.READY;
			END_IF
			IF(TransferType.1) THEN // TransferType =2 or 3
				HoBusy := FunctionRegistry[Param.reFunctionNumber].Zone[i].refZoneData.TransportControlData.eHandOverState <> E_HandOverState.IDLE AND
						  FunctionRegistry[Param.reFunctionNumber].Zone[i].refZoneData.TransportControlData.eHandOverState <> E_HandOverState.READY;			
			END_IF
		END_IF
	END_IF
	
	//Quit if busy
	IF(ToBusy OR HoBusy) THEN
		_M_TransferBusy:=TRUE;
		RETURN;
	END_IF
	
END_FOR
END_METHOD

END_FUNCTION_BLOCK

// ---- 20_Product/20_ProBox/22_ProMove/03_Controls/12_MotionPickAndDeposit/FB_DriveMover.TcPOU
FUNCTION_BLOCK FB_DriveMover
VAR_INPUT	 
	ErrorPending				 : BOOL; //Error active from element
	DisableEnableDrive			 : BOOL; // Request to turn off EnableDrive signal to Motion Freq. inveter when positioning finished.
	ElementOperationState		 : ST_PositionState; //Which state the element is in
	DriveCFG					 : ST_CFG_MPD_Drive; //Parameters to set up motion behaviour
	ManualControl				 : ST_MoviDriveManual; //Inputs located on shuttle
	EmgStopAxisTrig				 : BOOL; //Request to stop movment with emergency ramp settings.			
	DriveInputs					 : REFERENCE TO ST_PDO_DriveIn; //Inputs from frequency inverter 
	SemiDriveControl			: ST_SemiDriveControl;
	
END_VAR
VAR_OUTPUT
	DriveOutputs				: ST_PDO_DriveOut;	//Outputs to frequency inverter		
	AxisMotionOutputHigh		: BYTE; //Outputs sent to motion
	AxisMotionOutputLow			: BYTE; //Outputs sent to motion
	EnableDrive					: BOOL := FALSE; // Send to I/O module to enable the frequency inverter
	ActPos						: LREAL; //Indication where the machine really is
	Ready						: BOOL; //Indication that the mover is ready for an new assignment
	Busy						: BOOL; //Indication that the mover has an assignment (Movement may be finialized but will still regulate position)
 	Done						: BOOL; //Indication that the mover has completed it's assignment
	Aborted						: BOOL; //Indication that the mover was aborted during positioning and that the position may not be valid
END_VAR

VAR_IN_OUT
	ErrorData					: ST_ErrorDataSet; //Send an error to the overlaying element
END_VAR

VAR
 fbDelayEnable					: TOF;	
 CommissioningMode				: BOOL; //Activated to enable to run locally on motion
 Counter						: INT; //Counter to toggle an live flag to motion
 TrigMotionCmd					: BOOL; //Trig flag for applying new motion settings.
 StopAxis						: BOOL; //An request to stop the Axis
 StartPositioningAbsolute 		: BOOL; //Request to positioning absolute
 PositionToGo					: DINT; //Where the absolute positioning should go
 OverrideSpeed					: INT; //Choose how many % of the speed to move in
 Velocity						: INT; //How many mm/s to move in max speed
 Acceleration					: INT; //How many mm/s2 to accelerate in
 Deceleration					: INT; //How many mm/s2 to deccalerate in
 Jerk							: LREAL; //The jerk sent to motion.	
 MC_PowerRequest				: BOOL; //Internal request to turn on MC_Power
 PTP_ErrorCode					: UDINT; //Point-to-point error code sent from motion
 fbReleaseBrake					: TON :=(PT:=T#1S); //Timer for releasing the brake
 fbDisableEnableDrive			: TON :=(PT:=T#3S); //Delay for turning off EnableDrive signal.
 PositioningState				: E_PositioningState; //Enum state machine for the mover
 Axis 							: AXIS_REF; //Motion axis
 fbMC_MoveAbsolute1				: MC_MoveAbsolute; //TwinCat motion fb
 fbMC_MoveAbsolute2				: MC_MoveAbsolute; //TwinCat motion fb
 fbMC_SemiDriveHalt				: MC_Halt;  //TwinCat motion fb
 fbMC_Power						: MC_Power; //TwinCat motion fb
 fbMC_ReadParam					: MC_ReadParameter; //TwinCat motion fb
 fbMC_StopAxis					: MC_Stop; //TwinCat motion fb
 fbMC_Reset						: MC_Reset; //TwinCat motion fb
 fbMC_Jog						: MC_Jog; //TwinCat motion fb
 fbMC_WriteBoolParameter		: MC_WriteBoolParameter; //TwinCat motion fb
 DriveError						: BOOL;	//Input from ABB or SEW Motion Driver
 DriveResetError				: BOOL; //Output to ABB or SEW Motion Driver
 DriveReady						: BOOL; //Input from ABB or SEW Motion Driver
 R_TrigHalt						: R_Trig();

END_VAR
VAR_TEMP
	ManualModeReq				: BOOL; //manual mode request	
END_VAR

// Call axis
Axis();
Axis.ReadStatus();
fbMC_Reset(Axis := Axis);
fbMC_StopAxis(Axis := Axis);
fbMC_MoveAbsolute1(Axis := Axis);
fbMC_MoveAbsolute2(Axis := Axis);
fbMC_SemiDriveHalt(Axis := Axis);
fbMC_Jog(Axis := Axis);
fbMC_WriteBoolParameter(Axis := Axis);


 
fbMC_Power(
	Enable			:=  DriveReady AND MC_PowerRequest,
	Enable_Positive := TRUE,
	Enable_Negative := TRUE,
	Override		:= OverrideSpeed,
	Axis			:= Axis);
	
//set Stop axis when executing fbMC_MoveAbsolute, or inhibit start new operation
IF(EmgStopAxisTrig OR ( PositioningState = E_PositioningState.POSITIONING_ABSOLUTE AND (ElementOperationState.eMode <> E_PositionMode.AUTO_MODE OR ElementOperationState.eState = E_PositionState.STOPPED))) THEN
	StopAxis := TRUE;
END_IF

//check and reset errors
_M_ErrorHandler(ErrorData);

//Timer for releasing brake
fbReleaseBrake(IN:=DriveReady AND fbDelayEnable.Q , PT:=DriveCFG.TimeReleaseBrake , Q=> , ET=> );
//By default reset Disable enable drive timer
fbDisableEnableDrive.IN:=FALSE;

//Manual mode request
IF(ElementOperationState.eMode = E_PositionMode.MANUAL_MODE) THEN
	ManualModeReq:=TRUE;
ELSIF(SemiDriveControl.SemiManualMode AND ElementOperationState.eMode = E_PositionMode.AUTO_MODE  AND ElementOperationState.eState = E_PositionState.STARTED) THEN				 
	ManualModeReq:=TRUE;	
ELSE
	ManualModeReq:=FALSE;
END_IF				 

ManualModeReq := (ElementOperationState.eMode = E_PositionMode.MANUAL_MODE) OR
				 (SemiDriveControl.SemiManualMode AND ElementOperationState.eMode = E_PositionMode.AUTO_MODE  AND ElementOperationState.eState = E_PositionState.STARTED);


R_TrigHalt(CLK:= SemiDriveControl.SemiAutoMode AND SemiDriveControl.SemiAutoHalt); //Semi Auto drive mode halted
	
 			 

CASE PositioningState OF
	
(******************************************************************************
INIT
********************************************************************************)	
	E_PositioningState.INIT:
		EnableDrive := FALSE;
		StopAxis := FALSE;
		MC_PowerRequest := TRUE;
		Aborted:=TRUE;
		TrigMotionCmd:=FALSE;
		M_DisableSoftLimit(Disable := FALSE); 			
		// Drive is ready
		IF fbMC_Power.Status THEN
			fbMC_MoveAbsolute1(Execute := FALSE,Axis := Axis);
			fbMC_MoveAbsolute2(Execute := FALSE,Axis := Axis);
			fbMC_SemiDriveHalt(Execute := FALSE,Axis := Axis);
			fbMC_StopAxis(Execute := FALSE,Axis := Axis);
				
			EnableDrive := FALSE;				
			PositioningState := E_PositioningState.STANDBY;

		ELSE
			Ready := FALSE;
		END_IF

(******************************************************************************
COMMISSIONING MODE
********************************************************************************)
	E_PositioningState.COMMISSIONING:
		IF CommissioningMode THEN 
			MC_PowerRequest:=TRUE;
			EnableDrive := TRUE;
		ELSE
			PositioningState := E_PositioningState.INIT;
		END_IF	
(******************************************************************************
STANDBY
********************************************************************************)	
	E_PositioningState.STANDBY:
		//EnableDrive := FALSE;
		TrigMotionCmd:=FALSE;
		M_DisableSoftLimit(Disable := FALSE); 		
		MC_PowerRequest := TRUE;	
		// Drive is ready
		IF CommissioningMode THEN
			PositioningState := E_PositioningState.COMMISSIONING;
		
		ELSIF ElementOperationState.eMode = E_PositionMode.AUTO_MODE AND NOT ManualModeReq AND NOT ErrorPending AND NOT StopAxis AND DriveReady THEN
			Ready := TRUE;
			fbDisableEnableDrive.IN:=TRUE;
			IF(fbDisableEnableDrive.Q) THEN				
				EnableDrive := FALSE;
			END_IF
			IF  (*NOT Busy AND*) Ready AND fbMC_Power.Status (*PowerOnRequest*) AND StartPositioningAbsolute THEN					
					PositioningState := E_PositioningState.POSITIONING_ABSOLUTE;
					TrigMotionCmd:=TRUE;
					StartPositioningAbsolute:=FALSE;
			END_IF
			
		ELSIF ManualModeReq THEN
			EnableDrive := FALSE;	
			Ready := FALSE;
			PositioningState := E_PositioningState.MANUAL_MODE;
	
		ELSE
			EnableDrive := FALSE;
			Ready := FALSE;			
			IF ErrorPending THEN
				PositioningState := E_PositioningState.ERROR;
			ELSIF(StopAxis) THEN
				F_SetError( ErrorType:= E_ErrorType.ERROR, 	
							ErrorParam:= 'Motion aborted (1)',  
							ErrorMsg:= E_ErrorConv.DRIVE_WARNING, 
							ErrorData:= ErrorData);
				PositioningState := E_PositioningState.ERROR;
			END_IF
		END_IF
		
(******************************************************************************
POSITIONING_ABSOLUTE
********************************************************************************)	
	// Positioning
	E_PositioningState.POSITIONING_ABSOLUTE:
		
		// Call absolute positioning
 		IF(TrigMotionCmd AND fbReleaseBrake.Q)THEN
			TrigMotionCmd:=FALSE;
			IF(NOT fbMC_MoveAbsolute1.Busy) THEN 							
				fbMC_MoveAbsolute1(
					Execute := TRUE,
					Position := PositionToGo,
					Velocity := Velocity,
					Acceleration := Acceleration,
					Deceleration := Deceleration,
					Jerk := Jerk,
					BufferMode := MC_Aborting,
					Axis := Axis);		
			ELSE
				fbMC_MoveAbsolute2(
					Execute := TRUE,
					Position := PositionToGo,
					Velocity := Velocity,
					Acceleration := Acceleration,
					Deceleration := Deceleration,
					Jerk := Jerk,
					BufferMode := MC_Aborting,
					Axis := Axis);
			END_IF						
		END_IF		
		fbMC_MoveAbsolute1.Execute:=FALSE;
		fbMC_MoveAbsolute2.Execute:=FALSE;	
		EnableDrive := TRUE;           
		Busy := TRUE;					
		
		// Axis has an error (alternative Check Axis.Error)
		IF fbMC_MoveAbsolute1.Error OR fbMC_MoveAbsolute2.Error OR fbMC_SemiDriveHalt.Error THEN							
			Ready := FALSE;
			IF(fbMC_MoveAbsolute1.Error) THEN PTP_ErrorCode := fbMC_MoveAbsolute1.ErrorID;END_IF
			IF(fbMC_MoveAbsolute2.Error) THEN PTP_ErrorCode := fbMC_MoveAbsolute2.ErrorID;END_IF
			IF(fbMC_SemiDriveHalt.Error) THEN PTP_ErrorCode := fbMC_SemiDriveHalt.ErrorID;END_IF
			PositioningState := E_PositioningState.ERROR;
				
		// Axis has to be stopped abrupt		
		ELSIF StopAxis OR ErrorPending THEN							
			fbMC_StopAxis(
				Execute 		:= TRUE,
				Deceleration	:= DriveCFG.MaxDriveParamAuto.Deceleration,
				Jerk			:= DriveCFG.MaxDriveParamAuto.Jerk,
				Axis 			:= Axis,
				ErrorID			=> PTP_ErrorCode);
				
			Ready := FALSE;
			PositioningState := E_PositioningState.STOPPING;
		END_IF
			
		//Halt movement (only possible in semi autoMode) (Stay in POSITIONING_ABSOLUTE state) and possible to apply new data to fbMC_MoveAbsolute		
		fbMC_SemiDriveHalt.Execute := FALSE;
		IF(R_TrigHalt.Q)THEN
			IF(NOT SemiDriveControl.SemiTrigMoveAbs) THEN				
				fbMC_SemiDriveHalt(
					Execute := TRUE,				
					Deceleration := Deceleration,
					Jerk := Jerk,				
					Axis := Axis);	
			ELSE
				TrigMotionCmd :=TRUE;	// ->trig fbMC_MoveAbsolute 
			END_IF				
			Ready := FALSE;
			Aborted:=TRUE;		
							
		END_IF
		
		
		// Positioning finished
		IF (fbMC_MoveAbsolute1.Done OR fbMC_MoveAbsolute2.Done OR fbMC_SemiDriveHalt.Done) AND Axis.Status.NotMoving AND NOT Axis.Status.HasJob THEN			
			Done := fbMC_MoveAbsolute1.Done OR fbMC_MoveAbsolute2.Done;
			PositioningState := E_PositioningState.POSITIONING_FINISHED;
		END_IF
		
		//Finishing up things when leaving state
		IF(PositioningState <> E_PositioningState.POSITIONING_ABSOLUTE) THEN
			fbMC_MoveAbsolute1(Execute := FALSE,Axis := Axis);
			fbMC_MoveAbsolute2(Execute := FALSE,Axis := Axis);
			TrigMotionCmd:=FALSE;
		END_IF
		

(******************************************************************************
POSITIONING_FINISHED
********************************************************************************)	
	E_PositioningState.POSITIONING_FINISHED:
	
		IF ErrorPending THEN
			PositioningState := E_PositioningState.ERROR;
					
		ELSIF NOT Done THEN
			Busy := FALSE;
			PositioningState := E_PositioningState.STANDBY;
		
		ELSIF PositionToGo <> Axis.NcToPlc.SetPos THEN
			Busy := FALSE;			
			Done := FALSE;			
			PositioningState := E_PositioningState.STANDBY;
			
		ELSIF ManualModeReq THEN
			Done := FALSE;
			Busy := FALSE;
			PositioningState := E_PositioningState.STANDBY;
			
		ELSIF DisableEnableDrive THEN
			fbDisableEnableDrive.IN:=TRUE;
			IF(fbDisableEnableDrive.Q) THEN				
				EnableDrive := FALSE;				
				MC_PowerRequest := FALSE;
				Busy := FALSE;
				Aborted:=TRUE;				
			END_IF
		ELSE
			//Aborted shall be set if the state is not POSITIONING_FINISHED or not POSITIONING_ABSOLUTE or not STANDBY
			//Aborted shall be cleared once the position is guarantied
			Aborted:=FALSE;	
		END_IF
		
		
(******************************************************************************
STOPPING
********************************************************************************)
	E_PositioningState.STOPPING:
		fbMC_StopAxis(Execute := FALSE,Axis := Axis);
		Aborted:=TRUE;
		//TrigMotionCmd:=FALSE;
		
		//Wait for MC_Stop to finalize
		IF NOT fbMC_StopAxis.Busy OR fbMC_StopAxis.Error THEN
			
			// Remove enable flag on an error (especially after emergency stop) this allows the inverter to engage immediately the brake
			EnableDrive := FALSE; 			
			//DriveOutputs.FCB_Instance := 1; // Disable final stage			
			IF(StopAxis AND NOT ErrorPending) THEN
				StopAxis := FALSE;
				F_SetError( ErrorType:= E_ErrorType.ERROR, 	
							ErrorParam:= 'Motion aborted (2)',  
							ErrorMsg:= E_ErrorConv.DRIVE_WARNING, 
							ErrorData:= ErrorData);
			END_IF
			Busy := FALSE;
			PositioningState := E_PositioningState.STANDBY;
		END_IF

(******************************************************************************
HALTING
********************************************************************************)
	E_PositioningState.HALTING:
		PositioningState := E_PositioningState.STANDBY;		
		
		
(******************************************************************************
ERROR
********************************************************************************)
	
	// Drive or PTP is in error state
	E_PositioningState.ERROR:
		fbMC_StopAxis(
					Execute := FALSE,
					Axis := Axis);
		// Update SetPointPosition to avoid LagDistanceError
		Axis.PlcToNc.ExtSetPos := Axis.NcToPlc.ActPos;
		MC_PowerRequest := FALSE;
		Busy := FALSE;
		StopAxis := FALSE;
		EnableDrive := FALSE;
		Aborted:=TRUE;
		IF ManualModeReq THEN 
			PositioningState := E_PositioningState.MANUAL_MODE;
		ELSIF NOT ErrorPending THEN
			PositioningState := E_PositioningState.STANDBY;
		END_IF
		
(******************************************************************************
Manual Mode
********************************************************************************)
	E_PositioningState.MANUAL_MODE:
	
		fbMC_Jog.Acceleration 	:= DriveCFG.MaxDriveParamMan.Acceleration;
		fbMC_Jog.Deceleration 	:= DriveCFG.MaxDriveParamMan.Deceleration;
		fbMC_Jog.Jerk 		   	:= DriveCFG.MaxDriveParamMan.Jerk;	
		fbMC_Jog.Velocity	   	:= DriveCFG.MaxDriveParamMan.Velocity;
		fbMC_Jog.Mode			:= MC_JOGMODE_CONTINOUS;		
		Aborted:=TRUE;
		
		
		//Disable soft limits in motion
		IF ManualControl.EmergencyDrive THEN
			M_DisableSoftLimit(Disable := TRUE); 
		ELSIF NOT ManualControl.EmergencyDrive THEN
			M_DisableSoftLimit(Disable := FALSE); 			
		END_IF
		
		IF ((ManualControl.DriveFwd OR ManualControl.DriveRev) AND (ManualControl.DriveRev <> ManualControl.DriveFwd))  THEN
			MC_PowerRequest := TRUE;
			EnableDrive := TRUE;
			IF fbReleaseBrake.Q THEN				
				fbMC_Jog.JogForward := ManualControl.DriveFwd;
				fbMC_Jog.JogBackwards := ManualControl.DriveRev;
			END_IF		
					
		ELSIF NOT fbMC_Jog.Busy THEN
			EnableDrive := FALSE;
			MC_PowerRequest := FALSE;
			fbMC_Jog.JogForward := FALSE;
			fbMC_Jog.JogBackwards := FALSE;	
	
		ELSE
			fbMC_Jog.JogForward := FALSE;
			fbMC_Jog.JogBackwards := FALSE;				
		END_IF
		
		
		IF NOT ManualModeReq THEN
			EnableDrive := FALSE;			
			StopAxis := FALSE;
			fbMC_Jog.JogForward := FALSE;
			fbMC_Jog.JogBackwards := FALSE;			
			PositioningState := E_PositioningState.STANDBY;
		END_IF		

		// Set an error if lag distance gets to big or speed to high
		IF ElementOperationState.eState <> E_PositionState.STARTED THEN // Do not log lag and overspeed when Estop SS1 is active (i.e. FALSE)
			IF ABS(Axis.NcToPlc.PosDiff) > 200 AND (PTP_ErrorCode <> 998 AND PTP_ErrorCode <> 999) THEN
				 EnableDrive := FALSE;
				 PTP_ErrorCode := 998;
			ELSIF ABS(Axis.NcToPlc.SetVelo) > (DriveCFG.MaxDriveParamMan.Velocity + 10) AND (PTP_ErrorCode <> 998 AND PTP_ErrorCode <> 999) THEN

				 EnableDrive := FALSE;
				 PTP_ErrorCode := 999; 
			END_IF
		END_IF
END_CASE

fbDelayEnable(PT:= T#500MS, IN := EnableDrive);
fbDisableEnableDrive();
M_OutputMapping();

METHOD PRIVATE _M_ABB_ACS880 : BOOL
VAR_INPUT
END_VAR
//InputMapping
DriveError := DriveInputs.ABB_ACS880_StatusWord.Fault;
DriveReady := (DriveInputs.ABB_ACS880_StatusWord.ReadyToOperate OR DriveInputs.ABB_ACS880_StatusWord.ReadyToSwitchOn) AND 
			   DriveInputs.ABB_ACS880_StatusWord.RemoteCtrl;

//OutputMapping
DriveOutputs.ABB_ACS880_ControlWord.Reset := DriveResetError;
DriveOutputs.ABB_ACS880_ControlWord.Off_1 := fbDelayEnable.Q;
DriveOutputs.ABB_ACS880_ControlWord.Run := EnableDrive;//fbDelayEnable.Q; //By disabling this delay, the brake was locked earlier
END_METHOD

METHOD PRIVATE _M_ErrorHandler : BOOL
VAR_IN_OUT
	ErrorData						: ST_ErrorDataSet; //Send an error to the overlaying element
END_VAR
VAR_INST
	PrevCycleErrorPending 			: BOOL;
END_VAR
VAR
	 AcknowledgeError				: BOOL;
END_VAR

IF(PrevCycleErrorPending = TRUE AND ErrorPending = FALSE) THEN
	AcknowledgeError:=TRUE;
END_IF


//check configuration.
IF DriveCFG.InverterType = E_DriveMoverInverterType.ABB_ACS880 THEN 
	_M_ABB_ACS880();
ELSIF DriveCFG.InverterType = E_DriveMoverInverterType.SEW_MovidriveB THEN 
	_M_SEW_MoviDriveB();
ELSE 
	F_SetError( ErrorType:= E_ErrorType.ERROR, 	
				ErrorParam:=('No inverter type selected in cfg'),  
				ErrorMsg:= E_ErrorConv.CONFIGURATION_ERROR, 
				ErrorData:= ErrorData);	
END_IF



//Input error from laser/encoder
IF (Axis.NcToPlc.ActPos <= 0) AND Axis.Status.Homed AND NOT ManualControl.EmergencyDrive THEN
	F_SetError( ErrorType:= E_ErrorType.ERROR, 	
				ErrorParam:=('Actual position not valid'),  
				ErrorMsg:= E_ErrorConv.INCORRECT_ENCODER_VALUE, 
				ErrorData:= ErrorData);	
END_IF
	

// PTP Error Handling
IF (Axis.Status.Error OR PTP_ErrorCode <> 0) AND NOT fbMC_Reset.Busy THEN
	IF  AcknowledgeError(*NOT ErrorPending*) OR PositioningState = E_PositioningState.MANUAL_MODE THEN
		fbMC_Reset(
			Execute := TRUE,
			Axis := Axis);
		PTP_ErrorCode := 0;
		
	ELSE
		IF Axis.Status.Error THEN
			F_SetError( ErrorType:= E_ErrorType.ERROR, 	
						ErrorParam:= CONCAT('PTP error: ' , UDINT_TO_STRING(Axis.Status.ErrorID)),  
						ErrorMsg:= E_ErrorConv.DRIVE_ERROR, 
						ErrorData:= ErrorData);
		ELSE
			F_SetError( ErrorType:= E_ErrorType.ERROR, 	
						ErrorParam:= CONCAT('PTP error: ' , UDINT_TO_STRING(PTP_ErrorCode)),  
						ErrorMsg:= E_ErrorConv.DRIVE_ERROR, 
						ErrorData:= ErrorData);
		END_IF
	 
	END_IF
ELSIF(fbMC_Reset.Done) THEN
	fbMC_Reset(
		Execute := FALSE,
		Axis := Axis);
END_IF


//Drive error handling
IF NOT ErrorPending THEN
	IF DriveError AND NOT DriveResetError THEN
	// If reset requested, true to reset drive, do not set error this clockcycle	
		DriveResetError := TRUE;
	ELSIF DriveError AND DriveResetError THEN 
			F_SetError( ErrorType:= E_ErrorType.ERROR, 	
						ErrorParam:= 'Error on inverter' , 
						ErrorMsg:= E_ErrorConv.DRIVE_ERROR, 
						ErrorData:= ErrorData);
	END_IF
ELSE 
	DriveResetError := FALSE;
END_IF


//Check remote control on ABB drive
IF DriveCFG.InverterType = E_DriveMoverInverterType.ABB_ACS880 THEN 
	IF NOT DriveInputs.ABB_ACS880_StatusWord.RemoteCtrl THEN 
			F_SetError( ErrorType:= E_ErrorType.ERROR, 	
						ErrorParam:= 'ABB in local control' , 
						ErrorMsg:= E_ErrorConv.DRIVE_ERROR, 
						ErrorData:= ErrorData);
	END_IF
END_IF

//store current ErrorPending signal
PrevCycleErrorPending := ErrorPending;
END_METHOD

METHOD PRIVATE _M_SEW_MoviDriveB : BOOL
VAR_INPUT
END_VAR
//InputMapping
DriveError := DriveInputs.SEW_MoviDriveStatusWord.InverterError;
DriveReady := DriveInputs.SEW_MoviDriveStatusWord.InverterReadyForOperation;
//OutputMapping
DriveOutputs.SEW_MovidriveControlWord.ResetError := DriveResetError;
DriveOutputs.SEW_MovidriveControlWord.EnableAndQuickStop := fbDelayEnable.Q;
DriveOutputs.SEW_MovidriveControlWord.EnableAndStop := fbDelayEnable.Q;
END_METHOD

METHOD M_DisableSoftLimit : BOOL
VAR_INPUT
		Disable		: BOOL;
END_VAR

// Disable MinSoftPosLimit
fbMC_WriteBoolParameter(
	Execute := TRUE,
	ParameterNumber := AxisEnMinSoftPosLimit,
	Value := NOT Disable,
	Axis := Axis);
// Disable MaxSoftPosLimit
fbMC_WriteBoolParameter(
	Execute := TRUE,
	ParameterNumber := AxisEnMaxSoftPosLimit,
	Value := NOT Disable,
	Axis := Axis);
	
IF fbMC_WriteBoolParameter.Done THEN
	fbMC_WriteBoolParameter.Execute := FALSE;
	M_DisableSoftLimit := TRUE;
ELSE
	M_DisableSoftLimit := FALSE;
END_IF
END_METHOD

METHOD M_Init : BOOL
VAR_INPUT
END_VAR
VAR 
END_VAR

	OverrideSpeed := 100;
	StartPositioningAbsolute := FALSE;
	EnableDrive := FALSE;
	Busy := FALSE;
	Done := FALSE;
	
	// Jog configuration
	fbMC_Jog.Acceleration := DriveCFG.MaxDriveParamMan.Acceleration;
	fbMC_Jog.Deceleration := DriveCFG.MaxDriveParamMan.Deceleration;
	fbMC_Jog.Jerk 		   := DriveCFG.MaxDriveParamMan.Jerk;
	
	fbMC_StopAxis(
		Execute 		:= TRUE,
		Deceleration	:= 400000,
		Jerk			:= 400000,
		Axis 			:= Axis);
		
	PositioningState := E_PositioningState.INIT;
END_METHOD

METHOD M_MoveAbsolute : BOOL
(**************************************************************************************
 * 	AUTHOR		Swisslog
 * 	LIBRARY		Mover
 * 	PURPOSE		Trigger the axis to move to the specified position.
 *	RELEASE		1.0.0
 * ------------------------------------------------------------------------------------
 * 	Revision History: 
 *
 * 	VERSION		DATE		INITIALS	DESCRIPTION
 *	0.1			18.06.2013	ahe			initial version
 **************************************************************************************)
VAR_INPUT
	mPosition		: DINT;
	mVelocity		: INT;
	mAcceleration	: INT;
	mDeceleration	: INT;
	mJerk			: LREAL;	

END_VAR
VAR_IN_OUT
	ErrorData		: ST_ErrorDataSet;
END_VAR
VAR
	IsValid_PositionToGo	: BOOL;	
    IsValid_Velocity		: BOOL;
    IsValid_Acceleration	: BOOL;
    IsValid_Deceleration	: BOOL;
    IsValid_Jerk			: BOOL;
END_VAR


IsValid_PositionToGo 	:= FALSE;
IsValid_Velocity		:= FALSE;
IsValid_Acceleration	:= FALSE;
IsValid_Deceleration	:= FALSE;
IsValid_Jerk			:= FALSE;

// Check if position is inside the limits
IF mPosition > DriveCFG.MaximumPosition THEN
			F_SetError( ErrorType:= E_ErrorType.ERROR, 	
						ErrorParam:= 'Requested position over config max pos' , 
						ErrorMsg:= E_ErrorConv.DRIVE_ERROR, 
						ErrorData:= ErrorData);	
						
ELSIF mPosition < DriveCFG.MinimumPosition THEN
			F_SetError( ErrorType:= E_ErrorType.ERROR, 	
						ErrorParam:= 'Requested position under config min pos' , 
						ErrorMsg:= E_ErrorConv.DRIVE_ERROR, 
						ErrorData:= ErrorData);		
ELSE
	IsValid_PositionToGo := TRUE; 
	PositionToGo := mPosition;
END_IF

// Check if velocity is inside the limit
IF mVelocity > DriveCFG.MaxDriveParamAuto.Velocity THEN
			F_SetError( ErrorType:= E_ErrorType.ERROR, 	
						ErrorParam:= 'Requested velocity over max' , 
						ErrorMsg:= E_ErrorConv.DRIVE_ERROR, 
						ErrorData:= ErrorData);		
ELSE 
	IsValid_Velocity := TRUE;
	Velocity := mVelocity;	
END_IF

// Check if acceleration is inside the limit
IF mAcceleration > DriveCFG.MaxDriveParamAuto.Acceleration THEN
			F_SetError( ErrorType:= E_ErrorType.ERROR, 	
						ErrorParam:= 'Requested accelration over max' , 
						ErrorMsg:= E_ErrorConv.DRIVE_ERROR, 
						ErrorData:= ErrorData);	
ELSE
	IsValid_Acceleration := TRUE;
	Acceleration := mAcceleration;						
END_IF

// Check if deceleration is inside the limit
IF mDeceleration > DriveCFG.MaxDriveParamAuto.Deceleration THEN
			F_SetError( ErrorType:= E_ErrorType.ERROR, 	
						ErrorParam:= 'Requested deceleration over max' , 
						ErrorMsg:= E_ErrorConv.DRIVE_ERROR, 
						ErrorData:= ErrorData);	
ELSE
	IsValid_Deceleration := TRUE;
	Deceleration := mDeceleration;						
END_IF

// Check if jerk is inside the limit
IF mJerk > DriveCFG.MaxDriveParamAuto.Jerk THEN
			F_SetError( ErrorType:= E_ErrorType.ERROR, 	
						ErrorParam:= 'Requested jerk over max' , 
						ErrorMsg:= E_ErrorConv.DRIVE_ERROR, 
						ErrorData:= ErrorData);	
ELSE
	IsValid_Jerk := TRUE;
	Jerk := mJerk;						
END_IF

// Drive is ready to start
IF (NOT Busy AND Ready AND PositioningState = E_PositioningState.STANDBY AND NOT StopAxis AND
	 ElementOperationState.eMode = E_PositionMode.AUTO_MODE  AND ElementOperationState.eState = E_PositionState.STARTED AND
	IsValid_PositionToGo AND IsValid_Velocity AND IsValid_Acceleration AND IsValid_Deceleration AND IsValid_Jerk) THEN
	M_MoveAbsolute := TRUE;
	StartPositioningAbsolute := TRUE;	
ELSE
	M_MoveAbsolute := FALSE;
	StartPositioningAbsolute := FALSE;	
END_IF
END_METHOD

METHOD M_OutputMapping : BOOL
VAR

END_VAR


(****************************************************************************************************
					Hardware
*****************************************************************************************************)
//Mapping of drive are done in method for the drive

ActPos											:= Axis.NcToPlc.ActPos;

(****************************************************************************************************
					Motion
*****************************************************************************************************)
Counter:=Counter+1;
AxisMotionOutputLow.0 := 1; // Bit 0 : Ready to switch on
AxisMotionOutputLow.1 := 1; // Bit 1 : Switched on
AxisMotionOutputLow.2 := 1; // Bit 2 : Operation enabled
AxisMotionOutputLow.3 := 0; // Bit 3 : Fault
AxisMotionOutputLow.4 := 0; // Bit 4 : reserved
AxisMotionOutputLow.5 := 1; // Bit 5 : reserved
AxisMotionOutputLow.6 := 0; // Bit 6 : Switch on disabled
AxisMotionOutputLow.7 := 0; // // Bit 7 : Warning
AxisMotionOutputHigh.0 := 0; // Bit 8 : reserved
AxisMotionOutputHigh.1 := 0; // Bit 9 : reserved
AxisMotionOutputHigh.2 := Counter.6; // Bit 10 : TxPDOToggle
AxisMotionOutputHigh.3 := 0; // Bit 11 : Internal limit active
AxisMotionOutputHigh.4 := 1; // Bit 12 : Drive follows the command value  (note since TC_MC2 version 3.3.39 this bit has to be set on order for the Driver to set enable signal)
AxisMotionOutputHigh.5 := 0; // Bit 13 : Input cycle counter
AxisMotionOutputHigh.6 := 0; // Bit 14 - 15 : reserved
AxisMotionOutputHigh.7 := 0; // Bit 14 - 15 : reserved
END_METHOD

END_FUNCTION_BLOCK

// ---- 20_Product/20_ProBox/22_ProMove/03_Controls/12_MotionPickAndDeposit/FB_EntryReqControl.TcPOU
FUNCTION_BLOCK FB_EntryReqControl
VAR_INPUT
	//NumberOfCabinetsUsed	: INT;		// configure once for the system	
	ElementData				: REFERENCE TO ST_ElementData; //reference to SC/VC element data
	MpdRequestDone			: BOOL;	//the request is processed, and entry position is reached
END_VAR	
VAR_IN_OUT	
	EntryReqPositions				: ARRAY [*] OF DINT; // the SC/VC entry position [mm] for each panel index
END_VAR
	
VAR_OUTPUT
	ActiveCabinetIndex	: INT:=-1;	//init to an invalid index
	EntryRequest		: BOOL; // Entry requests. False = No requests pending, TRUE = Request pending or request active.
	EntryRequestCompl	: BOOL; // Entry request is completed and VC/Shuttle is in correct position.	
	EntryPosition		: DINT;	// The entry position [mm] of the level from where the entry is requested	
END_VAR
VAR CONSTANT
	ENTRY_REQ_MEM_BUFFER_MAX : INT :=100;
END_VAR
VAR
	_EntryState			: INT;//ARRAY[MIN_ENTRY_INDEX..MAX_ENTRY_INDEX] OF INT;
	_WaitForExternalDev	: BOOL; //wait in pending state for an external device
	_ActiveIndex		: INT;
	_RequestedPosition	: DINT;
	_EntryReqAbortMem	: ARRAY[0..ENTRY_REQ_MEM_BUFFER_MAX] OF BOOL; //Entry request abort memory buffer. 100 panels should be enouth

END_VAR

METHOD M_AbortEntryRequest : BOOL
VAR_INPUT
	CabinetIndex			: INT;		// the index of the cabinet
	Value					: BOOL;		//
END_VAR

IF(CabinetIndex>ENTRY_REQ_MEM_BUFFER_MAX) THEN	//outside max index
	RETURN;
ELSE
	_EntryReqAbortMem[CabinetIndex] := Value;
END_IF
END_METHOD

METHOD PUBLIC M_RegisterEntryRequest : BOOL
VAR_INPUT
	TriggEntryReq			: BOOL;		// Positive edge trigs an entry request
	CabinetIndex			: INT;		// the index of the cabinet
END_VAR

VAR CONSTANT

	STATE_IDLE 				: INT:=0;	// Wait for Enter request
	STATE_PENDING			: INT:=1;	// wait for SC/VC to move towards the entry position
	STATE_ACTIVE			: INT:=2;	// Entry position is reached, wait for key to turn back to Auto	
	STATE_DONE				: INT:=3;
END_VAR
VAR
	AbortEntryReq			: BOOL;
END_VAR

IF(NOT __ISVALIDREF(ElementData)) THEN
	RETURN;
END_IF

IF(EntryReqPositions[CabinetIndex]<=0) THEN //invalid position
	RETURN;
END_IF

AbortEntryReq := _EntryReqAbortMem[CabinetIndex];

//
CASE _EntryState OF
	STATE_IDLE:
		_ActiveIndex:=-1; //invalid index.
		IF(TriggEntryReq AND NOT AbortEntryReq AND
		   ElementData.OperationState.eMode = E_PositionMode.AUTO_MODE AND ElementData.OperationState.eState = E_PositionState.STARTED AND
		   LOWER_BOUND(EntryReqPositions,1)<=CabinetIndex AND UPPER_BOUND(EntryReqPositions,1)>=CabinetIndex)  THEN
					
			_EntryState := _EntryState+1;
			_ActiveIndex := CabinetIndex;
			_WaitForExternalDev :=FALSE;
			_RequestedPosition := EntryReqPositions[CabinetIndex];						 
		END_IF
				
	STATE_PENDING: //Entry State requested, wait for the SC/VC to move to the entry position	
		IF(MpdRequestDone AND NOT _WaitForExternalDev) THEN			
			_EntryState := _EntryState+1;
		END_IF
		
	STATE_ACTIVE:	//Wait user to turn back switch from entry request to auto mode
		IF((NOT TriggEntryReq AND CabinetIndex = _ActiveIndex) OR AbortEntryReq) THEN
			_EntryState := _EntryState+1;			
		END_IF
	
	STATE_DONE:
		_RequestedPosition := 0;		
		_EntryState:= STATE_IDLE;
END_CASE


//set outputs
EntryRequest		:= _EntryState=STATE_ACTIVE OR _EntryState=STATE_PENDING;
EntryRequestCompl	:= _EntryState=STATE_ACTIVE; //Request is completed.
ActiveCabinetIndex 	:= _ActiveIndex;
EntryPosition		:= _RequestedPosition;
END_METHOD

METHOD PUBLIC M_WaitForExternalDevice : BOOL
VAR_INPUT
	WaitForExternalDevice	: BOOL;		// wait in Entry pending state for an external device
	CabinetIndex			: INT;		// the index of the cabinet
END_VAR

IF(CabinetIndex=_ActiveIndex) THEN
	_WaitForExternalDev:= WaitForExternalDevice;
END_IF
END_METHOD

END_FUNCTION_BLOCK

// ---- 20_Product/20_ProBox/22_ProMove/03_Controls/12_MotionPickAndDeposit/FB_MPD_Control.TcPOU
//FB Motion Pickup n Deposit control
FUNCTION_BLOCK FB_MPD_Control
(**************************************************************************************
 * 	Application		:	BoxControl Framework
 *	Revision		:	$Revision:  $
 *	Revision date	:	$Date: $
 *	Last changed by	:	$Author: $
 *	URL				:	$URL: $
 *
 *	Purpose			:	Motion Pickup and Deposit (MPD) Functionality with one or two conveyors (A&B).
 *
 * ------------------------------------------------------------------------------------
 *	Copyright Swisslog [IP AG], Switzerland. All rights reserved.
 * 
 * ------------------------------------------------------------------------------------
 *	
 * 	Revision History: 
 *
 * 	VERSION			DATE			INITIALS			DESCRIPTION
 *
 **************************************************************************************)
VAR_INPUT
	MPD_Config				: ST_CFG_MotionPickupDeposit; 
	HW_Inputs		 		: ST_HW_InputsMPD; // Hardware inputs
	HW_Inputs_ManControl	: ST_HW_InputsManControl; // Hardware inputs manual control
	CtrlIn					: ST_CtrlInMPD_Control;
	ElementData				: REFERENCE TO ST_ElementData;
	FunctionOverides		: ARRAY[1..GVL_MPD.MAXPDs] OF BOOL; // internal data for function overrides, set by M_OverrridePickup
	IgnoreDepositCheck		: ARRAY[1..GVL_MPD.MAXPDs] OF BOOL; // internal data for disable conditions met for deposit functions, set by M_SetIgnoreDepositConditions
	OverhangData			: ARRAY[1..GVL_MPD.MAXPDs] OF BOOL; // internal data for function overrides, set by M_SetOverhangSensor
	ConvBrake				: ARRAY [1..2] OF BOOL; //Brake for conveyor A..B applied
	EmergencyStop			: BOOL; //Stop movment with emergency ramp profile.	
END_VAR                     	
                            	
VAR_OUTPUT
	HW_Outputs				: ST_HW_OutputsMPD;
	CtrlOut					: ST_CtrlOutMPD_Control;
	FunctionInterface		: ST_FunctionInterface;	// MPD conveyor drive request to element
	//MotionRunning			: BOOL; //True if motion is active and shuttle car / Lift is moving
END_VAR                     	
                            	
VAR		
	fbMPDPriority			: FB_MPD_PriorityControl;	//controls the prioirty and check conditions for pickup and deposit
	fbMPDMover				: FB_DriveMover; 		//Handlings moving of the shuttle
		
	//Private globals	
	_MPD					: ST_MPD;	// MPD data container.
	_MPDlInitDone			: BOOL;		// MPD (Motion Pickup and Deposit) control initializ complete.
	_EntryReqActive			: BOOL;		// Entry mode pending, request was activated by operator
	_EntryModeActive		: BOOL; 	// Entry door open mode active, request is finished	
	_AutoAdjustVcHeight		: ST_AutoAdjustVcHeight; //structure for auto height compensation used only for VC type
	_DebugPrint				: BOOL;
END_VAR



(**************************************************************************************************************
   Initialization
***************************************************************************************************************)
A_Init();



(**************************************************************************************************************
   Reset Error
***************************************************************************************************************)

F_ResetError(Reset 	  := FALSE,	ErrorData := ElementData.ErrorData.ErrorDataSet[3]); //Used for EndLimit 	
F_ResetError(Reset 	  := FALSE,	ErrorData := ElementData.ErrorData.ErrorDataSet[4]); //Used in Mover control	
F_ResetError(Reset 	  := FALSE,	ErrorData := ElementData.ErrorData.ErrorDataSet[5]); //Used in Motion and drive
F_ResetError(Reset 	  := FALSE,	ErrorData := ElementData.ErrorData.ErrorDataSet[6]); //used for overhang sensor check and EndLimit
F_ResetError(Reset 	  := FALSE,	ErrorData := ElementData.ErrorData.ErrorDataSet[7]); //Used in shuttle state control
F_ResetError(Reset 	  := FALSE,	ErrorData := ElementData.ErrorData.ErrorDataSet[8]); //Used in init


IF(_MPDlInitDone) THEN 
	(**************************************************************************************************************
		Run the priority controller always
	***************************************************************************************************************)
	fbMPDPriority(	ConfigPDs:=MPD_Config.ConvCFG,
					CvAFunctionNumber:= _MPD.CV[1].CvFuncNumber, 
					CvBFunctionNumber:= _MPD.CV[2].CvFuncNumber, 
					OverrideFunctions:= FunctionOverides,
					IgnoreDepositCheck:=IgnoreDepositCheck,
					MPD_Type         := MPD_Config.MPD_Type);
	
	(**************************************************************************************************************
	   Check overhang senors on Shuttle car and on adjacent functions
	***************************************************************************************************************)
	_M_CheckOverhangSensors();	
	
		
	(**************************************************************************************************************
	   Handle shuttle/VC conveyors
	***************************************************************************************************************)
	_M_SemiDriveControl();
	_M_MPD_Mover();
	_M_MPD_States();
	_M_MPD_CvStates(GVL_MPD.CV_A);
	_M_MPD_CvStates(GVL_MPD.CV_B);
	
			
	(**************************************************************************************************************
	   Output mapping
	***************************************************************************************************************)
	A_OutputMapping();	
	
	IF(ProBoxSystem.EMULATION_ENABLED) THEN
		_M_Emulation(MotionRunning:=CtrlOut.MotionRunning);	 
	END_IF
END_IF

//When picking/deposit pallets on the vertical conveyor and heavy loaded pallets moves in or moves out to/from VC the lifting unit will move up/down.
//This will apply stress is to the vc lifting unit and should be avoided by move UP a few mm when takeover pallet, and move DOWN a few mm when handover a pallet.
METHOD PRIVATE _M_AutoAdjustVCHeight : DINT
VAR_INPUT
	PickupActive	: BOOL;
	DepositActive	: BOOL;
	ResetAdjustment	: BOOL;
	ReturnAdjustedValue : BOOL;
END_VAR


VAR_INST
	HeightAdjusted		:BOOL;
	HeightAdjustedValue	: DINT;
END_VAR

//set default return value
_M_AutoAdjustVCHeight:=0;

//Auto Adjust height is only valid for Vertical conveyor type
IF(MPD_Config.MPD_Type	<> E_MotionPD_Type.E_VerticalCv) THEN
	RETURN;  
END_IF

IF(ResetAdjustment) THEN
	HeightAdjusted:=FALSE;	
	HeightAdjustedValue :=0;
	RETURN;	
END_IF


IF(ReturnAdjustedValue) THEN
	_M_AutoAdjustVCHeight:=HeightAdjustedValue;
	RETURN;
END_IF

IF(HeightAdjusted) THEN
	RETURN;
END_IF



// check occupied sensors on VC conveyor A and B

//When VC Taking over pallet...
IF(	PickupActive AND NOT DepositActive (*AND NOT F_PB_GetTransportControlDataRef(_MPD.CV[1].CvFuncNumber,1).Occupied*)) THEN
	IF( _AutoAdjustVcHeight.PickupCondition) THEN		
		_M_AutoAdjustVCHeight := _AutoAdjustVcHeight.PickupAdjustment;
		HeightAdjustedValue	:= _M_AutoAdjustVCHeight;
		HeightAdjusted:=TRUE;
	END_IF 
 END_IF

//When VC handing over pallet...
 IF( DepositActive AND NOT PickupActive (*AND F_PB_GetTransportControlDataRef(_MPD.CV[1].CvFuncNumber,1).Occupied*)) THEN	 
	 IF(_AutoAdjustVcHeight.DepositCondition) THEN
		_M_AutoAdjustVCHeight := _AutoAdjustVcHeight.DepositAdjustment;
		HeightAdjustedValue	:= _M_AutoAdjustVCHeight;
		HeightAdjusted:=TRUE;
	END_IF
 END_IF
END_METHOD

METHOD PRIVATE _M_CheckOverhangSensors
VAR
	i,j:INT;
	//OH_SensorVal 	: ARRAY [GVL_MPD.CV_A..GVL_MPD.CV_B] OF BOOL;
	TransferingTU	: ARRAY [GVL_MPD.CV_A..GVL_MPD.CV_B] OF BOOL; // internal variable used to determine if an pickup or deposit is currently ongoing
END_VAR

VAR_INST
	OH_SensorSide	: ARRAY [GVL_MPD.CV_A..GVL_MPD.CV_B] OF E_PickupDepositSide;
	AdjacentFunction: ARRAY [GVL_MPD.CV_A..GVL_MPD.CV_B] OF E_FunctionNumber;	
	OH_TestStart : ARRAY [GVL_MPD.CV_A..GVL_MPD.CV_B] OF BOOL;
	OH_TestEnd : ARRAY [GVL_MPD.CV_A..GVL_MPD.CV_B] OF BOOL;
	OH_TestCarOk : ARRAY [GVL_MPD.CV_A..GVL_MPD.CV_B] OF BOOL;
	OH_TestAdjacentSideOk : ARRAY [GVL_MPD.CV_A..GVL_MPD.CV_B] OF BOOL;
END_VAR
// Check overhang sensors
// 1. Check overhang sensors on Shuttle car / Vertical Conveyor
// 2. Check overhang sensors on conveyours connected to shuttle car Shuttle car / Vertical Conveytor
// 3. Check that overhang sensors is blocked during transport, just to make sure propper connection/setup etc


IF(	NOT _MPDlInitDone OR	ElementData.OperationState.eMode = E_PositionMode.MANUAL_MODE OR ElementData.OperationState.eState = E_PositionState.STOPPED) THEN	
	RETURN; //No not set over hang sensor error
END_IF

// Determine if an transfer is currently ongoing.
FOR i := GVL_MPD.CV_A TO GVL_MPD.CV_B BY 1 DO
	IF( _MPD.CV[i].State = E_MPD_CvStates.E_CV_PICKUP OR _MPD.CV[i].State = E_MPD_CvStates.E_CV_DEPOSIT) THEN
		TransferingTU[i]:=TRUE; //Transfer of TU is pending
	END_IF
END_FOR


// --------------------------------------------------------------------------------------
// 1.
// Check overhang sensors on shuttle car, but during transfer, the OH sensor on the transfering side shall not be considered.
// Get the side where the trasnfer is 
// Allow overhang sensor on the side where the transfer to toggle during transport. the other overhang sensor is to be used as "second" stop sensor just in case...
FOR i := GVL_MPD.CV_A TO GVL_MPD.CV_B BY 1 DO
	IF(_MPD.CV[i].State = E_MPD_CvStates.E_CV_PICKUP) THEN
		OH_SensorSide[i] := M_GetConveyorDirection(_MPD.CV[i].PickupFuncNumber); //Get the Pickup  side -> ignore overhang sensor on that side	
	ELSIF(_MPD.CV[i].State = E_MPD_CvStates.E_CV_DEPOSIT) THEN
		OH_SensorSide[i] := M_GetConveyorDirection(_MPD.CV[i].DepositFuncNumber); //Get the Pickup  side -> ignore overhang sensor on that side
	END_IF
END_FOR
	 
//Perform actual check
FOR i := GVL_MPD.CV_A TO GVL_MPD.CV_B BY 1 DO
	IF( _MPD.CV[i].Enabled AND 
		((HW_Inputs.Conv[i].SensorOverhangLeft = FALSE AND (OH_SensorSide[i] = E_PickupDepositSide.RightSide OR NOT TransferingTU[i])) OR   
		  (HW_Inputs.Conv[i].SensorOverhangRight = FALSE AND (OH_SensorSide[i] = E_PickupDepositSide.LeftSide OR NOT TransferingTU[i]))))THEN
		F_SetError( ErrorType:= E_ErrorType.ERROR, 	
					ErrorParam:= CONCAT('OverHangSensor: ',F_GetFunctionName(_MPD.CV[i].CvFuncNumber, 1(*zone one*))) , 
					ErrorMsg:= E_ErrorConv.INCORRECT_SENSOR_SIGNAL, ErrorData:= ElementData.ErrorData.ErrorDataSet[6]);
	END_IF
END_FOR



// --------------------------------------------------------------------------------------
// 2.
// Check overhang sensor on adjacent functions (ie pickup or deposit functions)
// This is ONLY needed while moving the car
IF( NOT TransferingTU[GVL_MPD.CV_A] AND NOT TransferingTU[GVL_MPD.CV_B]) THEN
	FOR i := 1 TO GVL_MPD.MAXPDs BY 1 DO	
		IF(MPD_Config.ConvCFG[i].eFunctionNumber <> E_FunctionNumber.F_BEGIN_FUNCTION AND NOT OverhangData[i])	THEN		
			F_SetError( ErrorType:= E_ErrorType.ERROR, 	
						ErrorParam:= CONCAT('OverHangSensor: ', F_GetFunctionName(MPD_Config.ConvCFG[i].eFunctionNumber, 0(*we dont know what zone it is, so we set the error to the funciton*))) , 
						ErrorMsg:= E_ErrorConv.INCORRECT_SENSOR_SIGNAL, ErrorData:= ElementData.ErrorData.ErrorDataSet[6]);										
		END_IF
	END_FOR
END_IF



// --------------------------------------------------------------------------------------
// 3.
// Check that overhang sensors are blocked during transport for conveyor A and B

FOR i := GVL_MPD.CV_A TO GVL_MPD.CV_B BY 1 DO
	IF(_MPD.CV[i].State = E_MPD_CvStates.E_CV_PICKUP) THEN 
		AdjacentFunction[i] := _MPD.CV[i].PickupFuncNumber;
	ELSIF(_MPD.CV[i].State = E_MPD_CvStates.E_CV_DEPOSIT) THEN 
		AdjacentFunction[i] := _MPD.CV[i].DepositFuncNumber;
	END_IF
END_FOR


// Start trig test. If CV is in correct state and drive is running (note, even if multiple zones, TransportActive reflects all zones) 
FOR i := GVL_MPD.CV_A TO GVL_MPD.CV_B BY 1 DO
	OH_TestStart[i] :=  OH_TestStart[i] OR (TransferingTU[i] AND F_PB_GetTransportControlDataRef(_MPD.CV[i].CvFuncNumber,i).TransportActive);		
END_FOR

//Montor sensors on shuttle car/Vertical conveyor, and register if it once where blocked
FOR i := GVL_MPD.CV_A TO GVL_MPD.CV_B BY 1 DO
	IF(OH_TestStart[i]) THEN
		OH_TestCarOk[i] := OH_TestCarOk[i] OR 
						  ((HW_Inputs.Conv[i].SensorOverhangLeft = FALSE AND (OH_SensorSide[i] = E_PickupDepositSide.LeftSide)) OR
						   (HW_Inputs.Conv[i].SensorOverhangRight = FALSE AND (OH_SensorSide[i] = E_PickupDepositSide.RightSide)));
	END_IF	
END_FOR

//Monitor sensor on the adjacent side function
FOR i := GVL_MPD.CV_A TO GVL_MPD.CV_B BY 1 DO
	IF(OH_TestStart[i]) THEN			
		FOR j := 1 TO GVL_MPD.MAXPDs BY 1 DO	
			IF(MPD_Config.ConvCFG[j].eFunctionNumber =AdjacentFunction[i] AND AdjacentFunction[i]<>E_FunctionNumber.F_BEGIN_FUNCTION)	THEN		
				OH_TestAdjacentSideOk[i] := OH_TestAdjacentSideOk[i] OR NOT OverhangData[j];											
			END_IF
		END_FOR
	END_IF
END_FOR

	   
//Check if transfer is finished.
FOR i := GVL_MPD.CV_A TO GVL_MPD.CV_B BY 1 DO
	OH_TestEnd[i] := OH_TestEnd[i] OR
					(OH_TestStart[i] AND  (_MPD.CV[i].State = E_MPD_CvStates.E_CV_OCCUPIED OR _MPD.CV[i].State = E_MPD_CvStates.E_CV_DONE));
END_FOR

FOR i := GVL_MPD.CV_A TO GVL_MPD.CV_B BY 1 DO
	IF(OH_TestEnd[i] AND NOT OH_TestCarOk[i]) THEN
		F_SetError( ErrorType:= E_ErrorType.ERROR, 	
					ErrorParam:= CONCAT('OverHang sensor was not blocked during transport: ',F_GetFunctionName(_MPD.CV[i].CvFuncNumber, 1(*zone one*))) , 
					ErrorMsg:= E_ErrorConv.INCORRECT_SENSOR_SIGNAL, ErrorData:= ElementData.ErrorData.ErrorDataSet[6]);
	END_IF
	
	IF(OH_TestEnd[i] AND NOT OH_TestAdjacentSideOk[i]) THEN
		F_SetError( ErrorType:= E_ErrorType.ERROR, 	
					ErrorParam:= CONCAT('Adjacent function OverHang sensor was not blocked during transport: ',F_GetFunctionName(AdjacentFunction[i], 0)) , 
					ErrorMsg:= E_ErrorConv.INCORRECT_SENSOR_SIGNAL, ErrorData:= ElementData.ErrorData.ErrorDataSet[6]);
	END_IF
END_FOR

	
 //Reset test flags (regardless if there was an error, since an error should only be trigged once and possible to acknowledge)
 FOR i := GVL_MPD.CV_A TO GVL_MPD.CV_B BY 1 DO
	IF(OH_TestEnd[i]) THEN 	
		OH_TestCarOk[i]:=OH_TestAdjacentSideOk[i]:=OH_TestStart[i]:=OH_TestEnd[i]:=FALSE;	
		AdjacentFunction[i]:=E_FunctionNumber.F_BEGIN_FUNCTION;			
	END_IF
END_FOR
END_METHOD

//Checks if a transport is complted. either handover or takeover is complete
METHOD PRIVATE _M_CheckTransportComplete : BOOL
VAR_INPUT
	CvState						: E_MPD_CvStates;
	CvIndex						: INT;		
END_VAR
VAR
	NumberOfZones				: INT:=1; // number of zones configured.
	i							: INT;
	IsOccupied					: BOOL;	
	isFree						: BOOL;
END_VAR
VAR_INST
	StabilityTimer				: ARRAY[GVL_MPD.CV_A..GVL_MPD.CV_B] OF TON();
END_VAR


//sanity checks
IF(NumberOfZones>conveyor.NUMBER_OF_ZONES_PER_FUNCTION) THEN RETURN;END_IF //error?


//Get number of zones configured.
IF(__ISVALIDREF(FunctionRegistry[_MPD.CV[CvIndex].CvFuncNumber].rSettingsFunction)) THEN
	NumberOfZones := FunctionRegistry[_MPD.CV[CvIndex].CvFuncNumber].rSettingsFunction.NumberOfZones;
END_IF


StabilityTimer[CvIndex].PT := SEL(NumberOfZones=1,T#1S,T#100MS);

CASE CvState OF
	
	//Pickup
	E_MPD_CvStates.E_CV_PICKUP:
	
	FOR i:=1 TO NumberOfZones DO
		IF( F_PB_GetTransportControlDataRef(_MPD.CV[CvIndex].CvFuncNumber,i).Occupied AND
			F_PB_GetTransportControlDataRef(_MPD.CV[CvIndex].CvFuncNumber,i).eTakeOverState <> E_TakeOverState.INTERRUPTED AND 
			F_PB_GetTransportControlDataRef(_MPD.CV[CvIndex].CvFuncNumber,i).eTakeOverState <> E_TakeOverState.STOP AND  
			(F_PB_GetTransportControlDataRef(_MPD.CV[CvIndex].CvFuncNumber,i).eTransportState = E_TransportState.OCCUPIED OR 
			 F_PB_GetTransportControlDataRef(_MPD.CV[CvIndex].CvFuncNumber,i).eTransportState = E_TransportState.SIMULTANEOUS_OCCUPIED)) THEN
			IsOccupied := TRUE;
		END_IF
	END_FOR
	
	StabilityTimer[CvIndex](IN:=IsOccupied); //needed when multiple zones configured
	
	//transport finished and brake are applied (not released)	
	_M_CheckTransportComplete:=StabilityTimer[CvIndex].Q AND IsOccupied AND NOT ConvBrake[CvIndex];
	
//Deposit -> Handover
	E_MPD_CvStates.E_CV_DEPOSIT:
		FOR i:=1 TO NumberOfZones DO
			IF( NOT F_PB_GetTransportControlDataRef(_MPD.CV[CvIndex].CvFuncNumber,i).Occupied AND
					F_PB_GetTransportControlDataRef(_MPD.CV[CvIndex].CvFuncNumber,i).eHandOverState <> E_HandOverState.INTERRUPTED AND
					F_PB_GetTransportControlDataRef(_MPD.CV[CvIndex].CvFuncNumber,i).eHandOverState <> E_HandOverState.STOP AND
					F_PB_GetTransportControlDataRef(_MPD.CV[CvIndex].CvFuncNumber,i).eTransportState <> E_TransportState.HANDOVER) THEN
				isFree:=TRUE;
			ELSE
				isFree:=FALSE;
				EXIT;
			END_IF
		END_FOR
			
		StabilityTimer[CvIndex](IN:=isFree); //needed when multiple zones configured
	
		//transport finished and brake are applied (not released)	
		_M_CheckTransportComplete:=StabilityTimer[CvIndex].Q AND isFree AND NOT ConvBrake[CvIndex];
		
	ELSE
		StabilityTimer[CvIndex](IN:=FALSE);
		
END_CASE
END_METHOD

METHOD PRIVATE _M_DebugPrint : BOOL
VAR_INPUT
	CvIndex	: INT; // 1=CV A, 2=CV B, 0=MPD Mover
	DbgMsg 	: STRING(System.DEBUGMESSAGELENGTH);
END_VAR

VAR_INST
	fbDebugMsg		: FB_DebugMsg; // Debug instance
	//DebugMsg		: T_MAXSTRING; // Debug msg
END_VAR

IF(CvIndex=0) THEN
	fbDebugMsg.M_SendInfoMsg(CONCAT('MPD: ', DbgMsg));
ELSIF(CvIndex<=GVL_MPD.CV_B) THEN
	fbDebugMsg.M_SendInfoMsg(CONCAT(CONCAT('MPD CV: ', GVL_MPD.CV_IxNAME[CvIndex]),CONCAT(': ', DbgMsg)));
ELSE
	fbDebugMsg.M_SendInfoMsg(DbgMsg);
END_IF
END_METHOD

METHOD PRIVATE _M_Emulation : BOOL
VAR_IN_OUT
	MotionRunning : BOOL;
END_VAR
VAR
	LastCyclePos : DINT;
END_VAR

IF(NOT ProBoxSystem.EMULATION_ENABLED) THEN
	RETURN;
END_IF

LastCyclePos := _MPD.ActualPosValue;

//emulate moving...
//consider speed?? MPD_Config.DriveCFG.DriveParameter[_MPD.DriveParameterIndex].Velocity/(1000/10(*10 ms CycleTime*))
IF(_MPD.RequestMove AND _M_IsErrorActive() = FALSE) THEN		
	IF( _MPD.ActualPosValue < _MPD.RequestPosValue) THEN _MPD.ActualPosValue := _MPD.ActualPosValue+4;	END_IF
	IF( _MPD.ActualPosValue > _MPD.RequestPosValue) THEN _MPD.ActualPosValue := _MPD.ActualPosValue-4;	END_IF		
					
	//check if desired position is within limits
	_MPD.Locked := M_CheckDesiredPosition(_MPD.RequestPosValue);
	
END_IF	

IF _EntryReqActive and _MPD.State = E_MPD_States.E_IDLE THEN 
	IF( _MPD.ActualPosValue < CtrlIn.RequestEntryPos) THEN _MPD.ActualPosValue := _MPD.ActualPosValue+4;	END_IF
	IF( _MPD.ActualPosValue > CtrlIn.RequestEntryPos) THEN _MPD.ActualPosValue := _MPD.ActualPosValue-4;	END_IF
	//check if desired position is within limits
	_MPD.Locked := M_CheckDesiredPosition(CtrlIn.RequestEntryPos);		
END_IF

MotionRunning := (_MPD.ActualPosValue <> LastCyclePos);
END_METHOD

//Get the pickup and deposit function from ShuttlePriority control FB_ShuttlePriorityControl
METHOD PRIVATE _M_GetPickupDepositFunctions: BOOL
VAR_INPUT
	CvIndex					: INT; // 1=A, 2=B	
	Verify					: BOOL; // set to true to check if actual pickup and deposit function still is the same
END_VAR
VAR
	rPrioFunctions			:REFERENCE TO ST_PrioFunctions;
END_VAR

IF(CvIndex = GVL_MPD.CV_A) THEN
	rPrioFunctions REF= fbMPDPriority.CV_A;
ELSIF(CvIndex = GVL_MPD.CV_B) THEN
	rPrioFunctions REF= fbMPDPriority.CV_B;
END_IF


//Sanity check
IF(NOT  __ISVALIDREF(rPrioFunctions)) THEN
	F_SetError(E_ErrorType.ERROR,'_M_GetPickupDepositFunctions bad reference',E_ErrorConv.SOFTWARE_ERROR,ElementData.ErrorData.ErrorDataSet[7]);
	RETURN;
END_IF


IF(Verify) THEN
	// check any position, as the priority may have been changed.
	_M_GetPickupDepositFunctions := (_MPD.CV[CvIndex].PickupFuncNumber = fbMPDPriority.CV_A.PickupFunctionNumber AND _MPD.CV[CvIndex].DepositFuncNumber = fbMPDPriority.CV_A.DepositFunctionNumber) OR
									(_MPD.CV[CvIndex].PickupFuncNumber = fbMPDPriority.CV_B.PickupFunctionNumber AND _MPD.CV[CvIndex].DepositFuncNumber = fbMPDPriority.CV_B.DepositFunctionNumber);
	RETURN;	
ELSIF( _MPD.CV[CvIndex].Enabled) THEN
	//revover...	
	IF( F_PB_GetTransportControlDataRef(_MPD.CV[CvIndex].CvFuncNumber,1).Occupied OR
		F_PB_GetTransportControlDataRef(_MPD.CV[CvIndex].CvFuncNumber,2).Occupied) THEN
		//recover after init etc..
		_MPD.CV[CvIndex].DepositFuncNumber := fbMPDPriority.M_GetDepositFunction(_MPD.CV[CvIndex].CvFuncNumber, 1, TRUE); 
		IF(_MPD.CV[CvIndex].DepositFuncNumber = E_FunctionNumber.F_BEGIN_FUNCTION) THEN
			_MPD.CV[CvIndex].DepositFuncNumber := fbMPDPriority.M_GetDepositFunction(_MPD.CV[CvIndex].CvFuncNumber, 2, TRUE);			
		END_IF 
		//IF(_MPD.CV[CvIndex].DepositFuncNumber = E_FunctionNumber.F_BEGIN_FUNCTION) //	-> no valid destination found
  
